LIN {X 0,Y 531.006,Z 455.967,A -85,B 0,C 180,E1 -4200.872,E2 -4200.872} C_VEL
LIN {X 0,Y 531.011,Z 455.964,A -85,B 0,C 180,E1 -4203.258,E2 -4203.258} C_VEL
LIN {X 0,Y 530.999,Z 456.014,A -85,B 0,C 180,E1 -4205.596,E2 -4205.596} C_VEL
LIN {X 0,Y 532.647,Z 464.711,A -85,B 0,C 180,E1 -4207.095,E2 -4207.095} C_VEL
LIN {X 0,Y 532.18,Z 482.462,A -85,B 0,C 180,E1 -4209.92,E2 -4209.92} C_VEL
LIN {X 0,Y 531.695,Z 501.444,A -85,B 0,C 180,E1 -4212.897,E2 -4212.897} C_VEL
LIN {X 0,Y 531.421,Z 515.316,A -85,B 0,C 180,E1 -4215.054,E2 -4215.054} C_VEL
LIN {X 0,Y 532.885,Z 524.969,A -85,B 0,C 180,E1 -4215.236,E2 -4215.236} C_VEL
LIN {X 0,Y 532.487,Z 624.081,A -85,B 0,C 180,E1 -4216.598,E2 -4216.598} C_VEL
LIN {X 0,Y 532.307,Z 637.145,A -85,B 0,C 180,E1 -4216.934,E2 -4216.934} C_VEL
LIN {X 0,Y 532.081,Z 649.714,A -85,B 0,C 180,E1 -4217.413,E2 -4217.413} C_VEL
LIN {X 0,Y 531.842,Z 661.515,A -85,B 0,C 180,E1 -4218.027,E2 -4218.027} C_VEL
LIN {X 0,Y 531.577,Z 672.421,A -85,B 0,C 180,E1 -4218.756,E2 -4218.756} C_VEL
LIN {X 0,Y 531.264,Z 682.786,A -85,B 0,C 180,E1 -4219.617,E2 -4219.617} C_VEL
LIN {X 0,Y 531.07,Z 691.257,A -85,B 0,C 180,E1 -4220.479,E2 -4220.479} C_VEL
LIN {X 0,Y 530.852,Z 700.523,A -85,B 0,C 180,E1 -4221.627,E2 -4221.627} C_VEL
LIN {X 0,Y 530.672,Z 707.981,A -85,B 0,C 180,E1 -4222.773,E2 -4222.773} C_VEL
LIN {X 0,Y 530.606,Z 713.97,A -85,B 0,C 180,E1 -4223.918,E2 -4223.918} C_VEL
LIN {X 0,Y 530.459,Z 718.708,A -85,B 0,C 180,E1 -4225.061,E2 -4225.061} C_VEL
LIN {X 0,Y 530.516,Z 722.337,A -85,B 0,C 180,E1 -4226.203,E2 -4226.203} C_VEL
LIN {X 0,Y 530.457,Z 724.213,A -85,B 0,C 180,E1 -4226.963,E2 -4226.963} C_VEL
LIN {X 0,Y 530.411,Z 725.631,A -85,B 0,C 180,E1 -4227.723,E2 -4227.723} C_VEL
LIN {X 0,Y 530.344,Z 727.258,A -85,B 0,C 180,E1 -4229.242,E2 -4229.242} C_VEL
LIN {X 0,Y 530.343,Z 727.497,A -85,B 0,C 180,E1 -4230.001,E2 -4230.001} C_VEL
LIN {X 0,Y 530.344,Z 727.313,A -85,B 0,C 180,E1 -4230.76,E2 -4230.76} C_VEL
LIN {X 0,Y 530.411,Z 725.758,A -85,B 0,C 180,E1 -4232.279,E2 -4232.279} C_VEL
LIN {X 0,Y 530.458,Z 724.396,A -85,B 0,C 180,E1 -4233.039,E2 -4233.039} C_VEL
LIN {X 0,Y 530.523,Z 721.517,A -85,B 0,C 180,E1 -4234.179,E2 -4234.179} C_VEL
LIN {X 0,Y 530.524,Z 717.614,A -85,B 0,C 180,E1 -4235.322,E2 -4235.322} C_VEL
LIN {X 0,Y 530.594,Z 712.029,A -85,B 0,C 180,E1 -4236.577,E2 -4236.577} C_VEL
LIN {X 0,Y 530.759,Z 705.018,A -85,B 0,C 180,E1 -4237.801,E2 -4237.801} C_VEL
LIN {X 0,Y 530.903,Z 696.833,A -85,B 0,C 180,E1 -4238.949,E2 -4238.949} C_VEL
LIN {X 0,Y 531.112,Z 688.547,A -85,B 0,C 180,E1 -4239.906,E2 -4239.906} C_VEL
LIN {X 0,Y 531.419,Z 678.357,A -85,B 0,C 180,E1 -4240.864,E2 -4240.864} C_VEL
LIN {X 0,Y 531.749,Z 666.673,A -85,B 0,C 180,E1 -4241.739,E2 -4241.739} C_VEL
LIN {X 0,Y 531.952,Z 655.511,A -85,B 0,C 180,E1 -4242.398,E2 -4242.398} C_VEL
LIN {X 0,Y 532.204,Z 642.456,A -85,B 0,C 180,E1 -4242.974,E2 -4242.974} C_VEL
LIN {X 0,Y 532.414,Z 629.216,A -85,B 0,C 180,E1 -4243.381,E2 -4243.381} C_VEL
LIN {X 0,Y 532.569,Z 616.016,A -85,B 0,C 180,E1 -4243.62,E2 -4243.62} C_VEL
LIN {X 0,Y 532.812,Z 523.746,A -85,B 0,C 180,E1 -4244.872,E2 -4244.872} C_VEL
LIN {X 0,Y 531.432,Z 515.327,A -85,B 0,C 180,E1 -4245.033,E2 -4245.033} C_VEL
LIN {X 0,Y 531.931,Z 493.174,A -85,B 0,C 180,E1 -4248.488,E2 -4248.488} C_VEL
LIN {X 0,Y 532.405,Z 474.148,A -85,B 0,C 180,E1 -4251.489,E2 -4251.489} C_VEL
LIN {X 0,Y 532.598,Z 463.987,A -85,B 0,C 180,E1 -4253.115,E2 -4253.115} C_VEL
LIN {X 0,Y 531.023,Z 455.965,A -85,B 0,C 180,E1 -4254.535,E2 -4254.535} C_VEL
LIN {X 0,Y 531.022,Z 455.969,A -85,B 0,C 180,E1 -4257.596,E2 -4257.596} C_VEL
LIN {X 0,Y 530.981,Z 455.968,A -85,B 0,C 180,E1 -4260.646,E2 -4260.646} C_VEL
LIN {X 0,Y 530.993,Z 455.97,A -85,B 0,C 180,E1 -4263.773,E2 -4263.773} C_VEL
LIN {X 0,Y 530.961,Z 455.967,A -85,B 0,C 180,E1 -4266.559,E2 -4266.559} C_VEL
LIN {X 0,Y 530.996,Z 455.967,A -85,B 0,C 180,E1 -4269.443,E2 -4269.443} C_VEL
LIN {X 0,Y 530.99,Z 455.964,A -85,B 0,C 180,E1 -4272.456,E2 -4272.456} C_VEL
LIN {X 0,Y 530.99,Z 455.97,A -85,B 0,C 180,E1 -4275.621,E2 -4275.621} C_VEL
LIN {X 0,Y 530.999,Z 455.961,A -85,B 0,C 180,E1 -4278.565,E2 -4278.565} C_VEL
LIN {X 0,Y 530.963,Z 455.972,A -85,B 0,C 180,E1 -4281.53,E2 -4281.53} C_VEL
LIN {X 0,Y 530.988,Z 455.964,A -85,B 0,C 180,E1 -4284.382,E2 -4284.382} C_VEL
LIN {X 0,Y 530.976,Z 455.966,A -85,B 0,C 180,E1 -4287.134,E2 -4287.134} C_VEL
LIN {X 0,Y 530.976,Z 455.973,A -85,B 0,C 180,E1 -4289.803,E2 -4289.803} C_VEL
LIN {X 0,Y 531.018,Z 455.961,A -85,B 0,C 180,E1 -4292.468,E2 -4292.468} C_VEL
LIN {X 0,Y 531.061,Z 456.072,A -85,B 0,C 180,E1 -4294.997,E2 -4294.997} C_VEL
LIN {X 0,Y 532.61,Z 464.294,A -85,B 0,C 180,E1 -4296.268,E2 -4296.268} C_VEL
LIN {X 0,Y 532.339,Z 481.085,A -85,B 0,C 180,E1 -4298.712,E2 -4298.712} C_VEL
LIN {X 0,Y 531.898,Z 502.756,A -85,B 0,C 180,E1 -4301.861,E2 -4301.861} C_VEL
LIN {X 0,Y 531.491,Z 524.306,A -85,B 0,C 180,E1 -4305.003,E2 -4305.003} C_VEL
LIN {X 0,Y 531.503,Z 525.159,A -85,B 0,C 180,E1 -4305.103,E2 -4305.103} C_VEL
LIN {X 0,Y 532.808,Z 533.582,A -85,B 0,C 180,E1 -4305.258,E2 -4305.258} C_VEL
LIN {X 0,Y 532.385,Z 632.475,A -85,B 0,C 180,E1 -4306.619,E2 -4306.619} C_VEL
LIN {X 0,Y 532.252,Z 643.791,A -85,B 0,C 180,E1 -4306.882,E2 -4306.882} C_VEL
LIN {X 0,Y 532.047,Z 656.313,A -85,B 0,C 180,E1 -4307.314,E2 -4307.314} C_VEL
LIN {X 0,Y 531.83,Z 669.019,A -85,B 0,C 180,E1 -4307.932,E2 -4307.932} C_VEL
LIN {X 0,Y 531.631,Z 679.052,A -85,B 0,C 180,E1 -4308.563,E2 -4308.563} C_VEL
LIN {X 0,Y 531.377,Z 687.856,A -85,B 0,C 180,E1 -4309.233,E2 -4309.233} C_VEL
LIN {X 0,Y 531.202,Z 695.315,A -85,B 0,C 180,E1 -4309.904,E2 -4309.904} C_VEL
LIN {X 0,Y 531.026,Z 702.592,A -85,B 0,C 180,E1 -4310.67,E2 -4310.67} C_VEL
LIN {X 0,Y 530.847,Z 710.181,A -85,B 0,C 180,E1 -4311.626,E2 -4311.626} C_VEL
LIN {X 0,Y 530.687,Z 716.517,A -85,B 0,C 180,E1 -4312.581,E2 -4312.581} C_VEL
LIN {X 0,Y 530.551,Z 722.563,A -85,B 0,C 180,E1 -4313.695,E2 -4313.695} C_VEL
LIN {X 0,Y 530.524,Z 726.919,A -85,B 0,C 180,E1 -4314.679,E2 -4314.679} C_VEL
LIN {X 0,Y 530.523,Z 730.899,A -85,B 0,C 180,E1 -4315.822,E2 -4315.822} C_VEL
LIN {X 0,Y 530.458,Z 733.85,A -85,B 0,C 180,E1 -4316.962,E2 -4316.962} C_VEL
LIN {X 0,Y 530.411,Z 735.354,A -85,B 0,C 180,E1 -4317.722,E2 -4317.722} C_VEL
LIN {X 0,Y 530.344,Z 736.92,A -85,B 0,C 180,E1 -4319.241,E2 -4319.241} C_VEL
LIN {X 0,Y 530.343,Z 737.208,A -85,B 0,C 180,E1 -4320,E2 -4320} C_VEL
LIN {X 0,Y 530.361,Z 736.404,A -85,B 0,C 180,E1 -4321.519,E2 -4321.519} C_VEL
LIN {X 0,Y 530.41,Z 735.49,A -85,B 0,C 180,E1 -4322.278,E2 -4322.278} C_VEL
LIN {X 0,Y 530.516,Z 732.244,A -85,B 0,C 180,E1 -4323.798,E2 -4323.798} C_VEL
LIN {X 0,Y 530.459,Z 728.685,A -85,B 0,C 180,E1 -4324.94,E2 -4324.94} C_VEL
LIN {X 0,Y 530.606,Z 725.794,A -85,B 0,C 180,E1 -4325.701,E2 -4325.701} C_VEL
LIN {X 0,Y 530.644,Z 720.318,A -85,B 0,C 180,E1 -4326.846,E2 -4326.846} C_VEL
LIN {X 0,Y 530.779,Z 713.434,A -85,B 0,C 180,E1 -4327.992,E2 -4327.992} C_VEL
LIN {X 0,Y 530.905,Z 706.468,A -85,B 0,C 180,E1 -4328.948,E2 -4328.948} C_VEL
LIN {X 0,Y 531.091,Z 699.912,A -85,B 0,C 180,E1 -4329.713,E2 -4329.713} C_VEL
LIN {X 0,Y 531.276,Z 691.104,A -85,B 0,C 180,E1 -4330.576,E2 -4330.576} C_VEL
LIN {X 0,Y 531.491,Z 682.944,A -85,B 0,C 180,E1 -4331.247,E2 -4331.247} C_VEL
LIN {X 0,Y 531.712,Z 673.503,A -85,B 0,C 180,E1 -4331.891,E2 -4331.891} C_VEL
LIN {X 0,Y 531.892,Z 664.443,A -85,B 0,C 180,E1 -4332.399,E2 -4332.399} C_VEL
LIN {X 0,Y 532.109,Z 653.571,A -85,B 0,C 180,E1 -4332.878,E2 -4332.878} C_VEL
LIN {X 0,Y 532.259,Z 642.616,A -85,B 0,C 180,E1 -4333.239,E2 -4333.239} C_VEL
LIN {X 0,Y 532.403,Z 631.966,A -85,B 0,C 180,E1 -4333.478,E2 -4333.478} C_VEL
LIN {X 0,Y 532.71,Z 532.707,A -85,B 0,C 180,E1 -4334.847,E2 -4334.847} C_VEL
LIN {X 0,Y 531.443,Z 524.939,A -85,B 0,C 180,E1 -4334.999,E2 -4334.999} C_VEL
LIN {X 0,Y 531.875,Z 505.036,A -85,B 0,C 180,E1 -4337.938,E2 -4337.938} C_VEL
LIN {X 0,Y 532.203,Z 485.232,A -85,B 0,C 180,E1 -4340.717,E2 -4340.717} C_VEL
LIN {X 0,Y 532.417,Z 472.579,A -85,B 0,C 180,E1 -4342.508,E2 -4342.508} C_VEL
LIN {X 0,Y 532.451,Z 463.714,A -85,B 0,C 180,E1 -4343.739,E2 -4343.739} C_VEL
LIN {X 0,Y 531.068,Z 455.96,A -85,B 0,C 180,E1 -4344.871,E2 -4344.871} C_VEL
LIN {X 0,Y 531.02,Z 455.963,A -85,B 0,C 180,E1 -4347.595,E2 -4347.595} C_VEL
LIN {X 0,Y 530.979,Z 455.97,A -85,B 0,C 180,E1 -4350.645,E2 -4350.645} C_VEL
LIN {X 0,Y 530.996,Z 455.968,A -85,B 0,C 180,E1 -4353.772,E2 -4353.772} C_VEL
LIN {X 0,Y 530.974,Z 455.968,A -85,B 0,C 180,E1 -4356.557,E2 -4356.557} C_VEL
LIN {X 0,Y 530.983,Z 455.972,A -85,B 0,C 180,E1 -4359.853,E2 -4359.853} C_VEL
LIN {X 0,Y 530.982,Z 455.967,A -85,B 0,C 180,E1 -4362.456,E2 -4362.456} C_VEL
LIN {X 0,Y 530.987,Z 455.97,A -85,B 0,C 180,E1 -4365.621,E2 -4365.621} C_VEL
LIN {X 0,Y 531.001,Z 455.962,A -85,B 0,C 180,E1 -4368.564,E2 -4368.564} C_VEL
LIN {X 0,Y 530.962,Z 455.973,A -85,B 0,C 180,E1 -4371.529,E2 -4371.529} C_VEL
LIN {X 0,Y 530.959,Z 455.968,A -85,B 0,C 180,E1 -4374.379,E2 -4374.379} C_VEL
LIN {X 0,Y 530.972,Z 455.971,A -85,B 0,C 180,E1 -4377.133,E2 -4377.133} C_VEL
LIN {X 0,Y 530.974,Z 455.971,A -85,B 0,C 180,E1 -4379.803,E2 -4379.803} C_VEL
LIN {X 0,Y 531.02,Z 455.963,A -85,B 0,C 180,E1 -4382.466,E2 -4382.466} C_VEL
LIN {X 0,Y 531.013,Z 456.03,A -85,B 0,C 180,E1 -4383.767,E2 -4383.767} C_VEL
LIN {X 0,Y 533.679,Z 467.602,A -85,B 0,C 180,E1 -4385.321,E2 -4385.321} C_VEL
LIN {X 0,Y 533.111,Z 489.338,A -85,B 0,C 180,E1 -4387.931,E2 -4387.931} C_VEL
LIN {X 0,Y 532.417,Z 514.942,A -85,B 0,C 180,E1 -4390.93,E2 -4390.93} C_VEL
LIN {X 0,Y 532.244,Z 523.261,A -85,B 0,C 180,E1 -4391.895,E2 -4391.895} C_VEL
LIN {X 0,Y 533.886,Z 534.58,A -85,B 0,C 180,E1 -4392.117,E2 -4392.117} C_VEL
LIN {X 0,Y 533.234,Z 661.903,A -85,B 0,C 180,E1 -4393.857,E2 -4393.857} C_VEL
LIN {X 0,Y 532.984,Z 676.417,A -85,B 0,C 180,E1 -4394.205,E2 -4394.205} C_VEL
LIN {X 0,Y 532.791,Z 690.417,A -85,B 0,C 180,E1 -4394.702,E2 -4394.702} C_VEL
LIN {X 0,Y 532.51,Z 702.779,A -85,B 0,C 180,E1 -4395.281,E2 -4395.281} C_VEL
LIN {X 0,Y 532.115,Z 715.658,A -85,B 0,C 180,E1 -4396.051,E2 -4396.051} C_VEL
LIN {X 0,Y 531.815,Z 727.295,A -85,B 0,C 180,E1 -4396.919,E2 -4396.919} C_VEL
LIN {X 0,Y 531.465,Z 738.305,A -85,B 0,C 180,E1 -4397.916,E2 -4397.916} C_VEL
LIN {X 0,Y 531.236,Z 747.698,A -85,B 0,C 180,E1 -4398.94,E2 -4398.94} C_VEL
LIN {X 0,Y 530.936,Z 756.55,A -85,B 0,C 180,E1 -4400.09,E2 -4400.09} C_VEL
LIN {X 0,Y 530.776,Z 765.028,A -85,B 0,C 180,E1 -4401.432,E2 -4401.432} C_VEL
LIN {X 0,Y 530.587,Z 771.859,A -85,B 0,C 180,E1 -4402.77,E2 -4402.77} C_VEL
LIN {X 0,Y 530.585,Z 777.957,A -85,B 0,C 180,E1 -4404.298,E2 -4404.298} C_VEL
LIN {X 0,Y 530.449,Z 781.441,A -85,B 0,C 180,E1 -4405.44,E2 -4405.44} C_VEL
LIN {X 0,Y 530.452,Z 784.831,A -85,B 0,C 180,E1 -4406.961,E2 -4406.961} C_VEL
LIN {X 0,Y 530.356,Z 786.834,A -85,B 0,C 180,E1 -4408.48,E2 -4408.48} C_VEL
LIN {X 0,Y 530.341,Z 787.5,A -85,B 0,C 180,E1 -4409.999,E2 -4409.999} C_VEL
LIN {X 0,Y 530.356,Z 786.837,A -85,B 0,C 180,E1 -4411.518,E2 -4411.518} C_VEL
LIN {X 0,Y 530.452,Z 784.838,A -85,B 0,C 180,E1 -4413.037,E2 -4413.037} C_VEL
LIN {X 0,Y 530.449,Z 781.45,A -85,B 0,C 180,E1 -4414.559,E2 -4414.559} C_VEL
LIN {X 0,Y 530.545,Z 776.571,A -85,B 0,C 180,E1 -4416.082,E2 -4416.082} C_VEL
LIN {X 0,Y 530.639,Z 770.059,A -85,B 0,C 180,E1 -4417.61,E2 -4417.61} C_VEL
LIN {X 0,Y 530.809,Z 762.81,A -85,B 0,C 180,E1 -4418.949,E2 -4418.949} C_VEL
LIN {X 0,Y 531.023,Z 753.83,A -85,B 0,C 180,E1 -4420.291,E2 -4420.291} C_VEL
LIN {X 0,Y 531.336,Z 744.403,A -85,B 0,C 180,E1 -4421.443,E2 -4421.443} C_VEL
LIN {X 0,Y 531.595,Z 733.963,A -85,B 0,C 180,E1 -4422.502,E2 -4422.502} C_VEL
LIN {X 0,Y 531.955,Z 722.441,A -85,B 0,C 180,E1 -4423.464,E2 -4423.464} C_VEL
LIN {X 0,Y 532.338,Z 709.642,A -85,B 0,C 180,E1 -4424.331,E2 -4424.331} C_VEL
LIN {X 0,Y 532.616,Z 697,A -85,B 0,C 180,E1 -4425.007,E2 -4425.007} C_VEL
LIN {X 0,Y 532.889,Z 683.114,A -85,B 0,C 180,E1 -4425.578,E2 -4425.578} C_VEL
LIN {X 0,Y 533.163,Z 668.658,A -85,B 0,C 180,E1 -4426.001,E2 -4426.001} C_VEL
LIN {X 0,Y 533.291,Z 654.28,A -85,B 0,C 180,E1 -4426.262,E2 -4426.262} C_VEL
LIN {X 0,Y 533.824,Z 533.283,A -85,B 0,C 180,E1 -4427.902,E2 -4427.902} C_VEL
LIN {X 0,Y 532.256,Z 523.34,A -85,B 0,C 180,E1 -4428.095,E2 -4428.095} C_VEL
LIN {X 0,Y 532.905,Z 496.157,A -85,B 0,C 180,E1 -4431.263,E2 -4431.263} C_VEL
LIN {X 0,Y 533.655,Z 471.16,A -85,B 0,C 180,E1 -4434.239,E2 -4434.239} C_VEL
LIN {X 0,Y 533.728,Z 467.421,A -85,B 0,C 180,E1 -4434.691,E2 -4434.691} C_VEL
LIN {X 0,Y 531.003,Z 455.969,A -85,B 0,C 180,E1 -4436.26,E2 -4436.26} C_VEL
LIN {X 0,Y 530.997,Z 455.964,A -85,B 0,C 180,E1 -4439.32,E2 -4439.32} C_VEL
LIN {X 0,Y 530.977,Z 455.967,A -85,B 0,C 180,E1 -4442.102,E2 -4442.102} C_VEL
LIN {X 0,Y 530.986,Z 455.963,A -85,B 0,C 180,E1 -4444.853,E2 -4444.853} C_VEL
LIN {X 0,Y 530.962,Z 455.967,A -85,B 0,C 180,E1 -4447.506,E2 -4447.506} C_VEL
LIN {X 0,Y 531.022,Z 455.965,A -85,B 0,C 180,E1 -4450.427,E2 -4450.427} C_VEL
LIN {X 0,Y 530.962,Z 455.966,A -85,B 0,C 180,E1 -4453.493,E2 -4453.493} C_VEL
LIN {X 0,Y 530.959,Z 455.972,A -85,B 0,C 180,E1 -4456.505,E2 -4456.505} C_VEL
LIN {X 0,Y 531.001,Z 455.96,A -85,B 0,C 180,E1 -4459.569,E2 -4459.569} C_VEL
LIN {X 0,Y 530.96,Z 455.972,A -85,B 0,C 180,E1 -4462.576,E2 -4462.576} C_VEL
LIN {X 0,Y 530.996,Z 455.96,A -85,B 0,C 180,E1 -4465.311,E2 -4465.311} C_VEL
LIN {X 0,Y 530.973,Z 455.965,A -85,B 0,C 180,E1 -4468.032,E2 -4468.032} C_VEL
LIN {X 0,Y 530.997,Z 455.967,A -85,B 0,C 180,E1 -4470.87,E2 -4470.87} C_VEL
LIN {X 0,Y 531.003,Z 455.962,A -85,B 0,C 180,E1 -4473.256,E2 -4473.256} C_VEL
LIN {X 0,Y 530.986,Z 455.962,A -85,B 0,C 180,E1 -4475.957,E2 -4475.957} C_VEL
LIN {X 0,Y 530.992,Z 455.962,A -85,B 0,C 180,E1 -4479.062,E2 -4479.062} C_VEL
LIN {X 0,Y 531.005,Z 455.965,A -85,B 0,C 180,E1 -4482.277,E2 -4482.277} C_VEL
LIN {X 0,Y 531.008,Z 455.96,A -85,B 0,C 180,E1 -4485.436,E2 -4485.436} C_VEL
LIN {X 0,Y 531.036,Z 455.963,A -85,B 0,C 180,E1 -4488.55,E2 -4488.55} C_VEL
LIN {X 0,Y 531.051,Z 455.955,A -85,B 0,C 180,E1 -4491.629,E2 -4491.629} C_VEL
LIN {X 0,Y 531.132,Z 455.953,A -85,B 0,C 180,E1 -4494.685,E2 -4494.685} C_VEL
LIN {X 0,Y 531.13,Z 455.944,A -85,B 0,C 180,E1 -4497.725,E2 -4497.725} C_VEL
LIN {X 0,Y 531.146,Z 455.95,A -85,B 0,C 180,E1 -4500.758,E2 -4500.758} C_VEL
LIN {X 0,Y 531.101,Z 455.948,A -85,B 0,C 180,E1 -4503.034,E2 -4503.034} C_VEL
LIN {X 0,Y 531.074,Z 455.955,A -85,B 0,C 180,E1 -4506.077,E2 -4506.077} C_VEL
LIN {X 0,Y 531.026,Z 455.959,A -85,B 0,C 180,E1 -4509.138,E2 -4509.138} C_VEL
LIN {X 0,Y 531.03,Z 455.962,A -85,B 0,C 180,E1 -4512.225,E2 -4512.225} C_VEL
LIN {X 0,Y 530.986,Z 455.963,A -85,B 0,C 180,E1 -4515.35,E2 -4515.35} C_VEL
LIN {X 0,Y 531.006,Z 455.959,A -85,B 0,C 180,E1 -4517.723,E2 -4517.723} C_VEL
LIN {X 0,Y 530.992,Z 455.965,A -85,B 0,C 180,E1 -4520.938,E2 -4520.938} C_VEL
LIN {X 0,Y 530.97,Z 455.97,A -85,B 0,C 180,E1 -4524.225,E2 -4524.225} C_VEL
LIN {X 0,Y 531.003,Z 455.966,A -85,B 0,C 180,E1 -4526.744,E2 -4526.744} C_VEL
LIN {X 0,Y 530.991,Z 455.962,A -85,B 0,C 180,E1 -4529.322,E2 -4529.322} C_VEL
LIN {X 0,Y 530.972,Z 455.968,A -85,B 0,C 180,E1 -4532.104,E2 -4532.104} C_VEL
LIN {X 0,Y 530.984,Z 455.968,A -85,B 0,C 180,E1 -4534.856,E2 -4534.856} C_VEL
LIN {X 0,Y 530.96,Z 455.965,A -85,B 0,C 180,E1 -4537.508,E2 -4537.508} C_VEL
LIN {X 0,Y 531.02,Z 455.967,A -85,B 0,C 180,E1 -4540.43,E2 -4540.43} C_VEL
LIN {X 0,Y 530.955,Z 455.967,A -85,B 0,C 180,E1 -4543.578,E2 -4543.578} C_VEL
LIN {X 0,Y 530.284,Z 456.057,A -85,B 0,C 180,E1 -4544.212,E2 -4544.212} C_VEL
LIN {X 0,Y 527.438,Z 456.413,A -85,B 0,C 180,E1 -4545.241,E2 -4545.241} C_VEL
LIN {X 0,Y 525.035,Z 456.713,A -85,B 0,C 180,E1 -4546.069,E2 -4546.069} C_VEL
LIN {X 0,Y 524.002,Z 456.84,A -85,B 0,C 180,E1 -4546.709,E2 -4546.709} C_VEL
LIN {X 0,Y 523.917,Z 456.847,A -85,B 0,C 180,E1 -4546.925,E2 -4546.925} C_VEL
LIN {X 0,Y 523.974,Z 456.839,A -85,B 0,C 180,E1 -4549.925,E2 -4549.925} C_VEL
LIN {X 0,Y 523.908,Z 456.847,A -85,B 0,C 180,E1 -4552.87,E2 -4552.87} C_VEL
LIN {X 0,Y 523.943,Z 456.842,A -85,B 0,C 180,E1 -4555.712,E2 -4555.712} C_VEL
LIN {X 0,Y 523.931,Z 456.848,A -85,B 0,C 180,E1 -4558.458,E2 -4558.458} C_VEL
LIN {X 0,Y 523.95,Z 456.844,A -85,B 0,C 180,E1 -4561.127,E2 -4561.127} C_VEL
LIN {X 0,Y 523.985,Z 456.842,A -85,B 0,C 180,E1 -4563.981,E2 -4563.981} C_VEL
LIN {X 0,Y 523.985,Z 456.933,A -85,B 0,C 180,E1 -4565.379,E2 -4565.379} C_VEL
LIN {X 0,Y 525.753,Z 466.105,A -85,B 0,C 180,E1 -4566.985,E2 -4566.985} C_VEL
LIN {X 0,Y 525.292,Z 482.605,A -85,B 0,C 180,E1 -4569.645,E2 -4569.645} C_VEL
LIN {X 0,Y 524.777,Z 501.605,A -85,B 0,C 180,E1 -4572.665,E2 -4572.665} C_VEL
LIN {X 0,Y 524.451,Z 515.395,A -85,B 0,C 180,E1 -4574.829,E2 -4574.829} C_VEL
LIN {X 0,Y 526.097,Z 525.449,A -85,B 0,C 180,E1 -4575.02,E2 -4575.02} C_VEL
LIN {X 0,Y 525.687,Z 623.589,A -85,B 0,C 180,E1 -4576.372,E2 -4576.372} C_VEL
LIN {X 0,Y 525.489,Z 636.208,A -85,B 0,C 180,E1 -4576.687,E2 -4576.687} C_VEL
LIN {X 0,Y 525.241,Z 649.671,A -85,B 0,C 180,E1 -4577.197,E2 -4577.197} C_VEL
LIN {X 0,Y 524.976,Z 660.656,A -85,B 0,C 180,E1 -4577.762,E2 -4577.762} C_VEL
LIN {X 0,Y 524.713,Z 671.91,A -85,B 0,C 180,E1 -4578.509,E2 -4578.509} C_VEL
LIN {X 0,Y 524.344,Z 682.423,A -85,B 0,C 180,E1 -4579.381,E2 -4579.381} C_VEL
LIN {X 0,Y 524.111,Z 691.886,A -85,B 0,C 180,E1 -4580.352,E2 -4580.352} C_VEL
LIN {X 0,Y 523.893,Z 699.65,A -85,B 0,C 180,E1 -4581.321,E2 -4581.321} C_VEL
LIN {X 0,Y 523.66,Z 707.249,A -85,B 0,C 180,E1 -4582.482,E2 -4582.482} C_VEL
LIN {X 0,Y 523.542,Z 714.234,A -85,B 0,C 180,E1 -4583.836,E2 -4583.836} C_VEL
LIN {X 0,Y 523.383,Z 718.899,A -85,B 0,C 180,E1 -4584.994,E2 -4584.994} C_VEL
LIN {X 0,Y 523.443,Z 722.463,A -85,B 0,C 180,E1 -4586.152,E2 -4586.152} C_VEL
LIN {X 0,Y 523.367,Z 724.313,A -85,B 0,C 180,E1 -4586.922,E2 -4586.922} C_VEL
LIN {X 0,Y 523.335,Z 725.709,A -85,B 0,C 180,E1 -4587.692,E2 -4587.692} C_VEL
LIN {X 0,Y 523.25,Z 727.316,A -85,B 0,C 180,E1 -4589.231,E2 -4589.231} C_VEL
LIN {X 0,Y 523.247,Z 727.551,A -85,B 0,C 180,E1 -4590.001,E2 -4590.001} C_VEL
LIN {X 0,Y 523.25,Z 727.369,A -85,B 0,C 180,E1 -4590.771,E2 -4590.771} C_VEL
LIN {X 0,Y 523.335,Z 725.831,A -85,B 0,C 180,E1 -4592.31,E2 -4592.31} C_VEL
LIN {X 0,Y 523.368,Z 724.489,A -85,B 0,C 180,E1 -4593.08,E2 -4593.08} C_VEL
LIN {X 0,Y 523.442,Z 721.651,A -85,B 0,C 180,E1 -4594.236,E2 -4594.236} C_VEL
LIN {X 0,Y 523.463,Z 717.811,A -85,B 0,C 180,E1 -4595.394,E2 -4595.394} C_VEL
LIN {X 0,Y 523.518,Z 712.761,A -85,B 0,C 180,E1 -4596.575,E2 -4596.575} C_VEL
LIN {X 0,Y 523.682,Z 706.637,A -85,B 0,C 180,E1 -4597.713,E2 -4597.713} C_VEL
LIN {X 0,Y 523.895,Z 698.849,A -85,B 0,C 180,E1 -4598.875,E2 -4598.875} C_VEL
LIN {X 0,Y 524.152,Z 689.17,A -85,B 0,C 180,E1 -4600.039,E2 -4600.039} C_VEL
LIN {X 0,Y 524.486,Z 679.066,A -85,B 0,C 180,E1 -4601.009,E2 -4601.009} C_VEL
LIN {X 0,Y 524.86,Z 667.864,A -85,B 0,C 180,E1 -4601.867,E2 -4601.867} C_VEL
LIN {X 0,Y 525.079,Z 656.426,A -85,B 0,C 180,E1 -4602.563,E2 -4602.563} C_VEL
LIN {X 0,Y 525.355,Z 644.892,A -85,B 0,C 180,E1 -4603.097,E2 -4603.097} C_VEL
LIN {X 0,Y 525.559,Z 632.511,A -85,B 0,C 180,E1 -4603.51,E2 -4603.51} C_VEL
LIN {X 0,Y 525.728,Z 619.999,A -85,B 0,C 180,E1 -4603.776,E2 -4603.776} C_VEL
LIN {X 0,Y 525.992,Z 524.359,A -85,B 0,C 180,E1 -4605.084,E2 -4605.084} C_VEL
LIN {X 0,Y 524.449,Z 515.252,A -85,B 0,C 180,E1 -4605.283,E2 -4605.283} C_VEL
LIN {X 0,Y 524.979,Z 494.705,A -85,B 0,C 180,E1 -4608.519,E2 -4608.519} C_VEL
LIN {X 0,Y 525.362,Z 478.073,A -85,B 0,C 180,E1 -4611.174,E2 -4611.174} C_VEL
LIN {X 0,Y 525.773,Z 466.631,A -85,B 0,C 180,E1 -4613.017,E2 -4613.017} C_VEL
LIN {X 0,Y 523.981,Z 456.843,A -85,B 0,C 180,E1 -4614.729,E2 -4614.729} C_VEL
LIN {X 0,Y 523.985,Z 456.847,A -85,B 0,C 180,E1 -4617.719,E2 -4617.719} C_VEL
LIN {X 0,Y 523.951,Z 456.844,A -85,B 0,C 180,E1 -4620.855,E2 -4620.855} C_VEL
LIN {X 0,Y 523.965,Z 456.846,A -85,B 0,C 180,E1 -4623.735,E2 -4623.735} C_VEL
LIN {X 0,Y 523.909,Z 456.846,A -85,B 0,C 180,E1 -4626.402,E2 -4626.402} C_VEL
LIN {X 0,Y 523.929,Z 456.843,A -85,B 0,C 180,E1 -4629.085,E2 -4629.085} C_VEL
LIN {X 0,Y 523.964,Z 456.842,A -85,B 0,C 180,E1 -4632.119,E2 -4632.119} C_VEL
LIN {X 0,Y 523.961,Z 456.841,A -85,B 0,C 180,E1 -4635.309,E2 -4635.309} C_VEL
LIN {X 0,Y 523.961,Z 456.837,A -85,B 0,C 180,E1 -4638.69,E2 -4638.69} C_VEL
LIN {X 0,Y 523.923,Z 456.844,A -85,B 0,C 180,E1 -4641.081,E2 -4641.081} C_VEL
LIN {X 0,Y 523.935,Z 456.849,A -85,B 0,C 180,E1 -4643.828,E2 -4643.828} C_VEL
LIN {X 0,Y 523.949,Z 456.84,A -85,B 0,C 180,E1 -4646.636,E2 -4646.636} C_VEL
LIN {X 0,Y 523.961,Z 456.843,A -85,B 0,C 180,E1 -4649.356,E2 -4649.356} C_VEL
LIN {X 0,Y 523.983,Z 456.839,A -85,B 0,C 180,E1 -4652.282,E2 -4652.282} C_VEL
LIN {X 0,Y 524.034,Z 456.99,A -85,B 0,C 180,E1 -4654.824,E2 -4654.824} C_VEL
LIN {X 0,Y 525.683,Z 465.511,A -85,B 0,C 180,E1 -4656.151,E2 -4656.151} C_VEL
LIN {X 0,Y 525.437,Z 479.564,A -85,B 0,C 180,E1 -4658.212,E2 -4658.212} C_VEL
LIN {X 0,Y 525.055,Z 497.625,A -85,B 0,C 180,E1 -4660.856,E2 -4660.856} C_VEL
LIN {X 0,Y 524.631,Z 518.142,A -85,B 0,C 180,E1 -4663.861,E2 -4663.861} C_VEL
LIN {X 0,Y 524.523,Z 525.245,A -85,B 0,C 180,E1 -4664.9,E2 -4664.9} C_VEL
LIN {X 0,Y 525.954,Z 534.643,A -85,B 0,C 180,E1 -4665.081,E2 -4665.081} C_VEL
LIN {X 0,Y 525.444,Z 633.269,A -85,B 0,C 180,E1 -4666.463,E2 -4666.463} C_VEL
LIN {X 0,Y 525.332,Z 646.029,A -85,B 0,C 180,E1 -4666.78,E2 -4666.78} C_VEL
LIN {X 0,Y 525.05,Z 659.504,A -85,B 0,C 180,E1 -4667.29,E2 -4667.29} C_VEL
LIN {X 0,Y 524.795,Z 671.704,A -85,B 0,C 180,E1 -4667.929,E2 -4667.929} C_VEL
LIN {X 0,Y 524.571,Z 681.798,A -85,B 0,C 180,E1 -4668.602,E2 -4668.602} C_VEL
LIN {X 0,Y 524.277,Z 692.414,A -85,B 0,C 180,E1 -4669.476,E2 -4669.476} C_VEL
LIN {X 0,Y 524.012,Z 702.751,A -85,B 0,C 180,E1 -4670.544,E2 -4670.544} C_VEL
LIN {X 0,Y 523.825,Z 710.34,A -85,B 0,C 180,E1 -4671.513,E2 -4671.513} C_VEL
LIN {X 0,Y 523.629,Z 717.75,A -85,B 0,C 180,E1 -4672.674,E2 -4672.674} C_VEL
LIN {X 0,Y 523.504,Z 723.712,A -85,B 0,C 180,E1 -4673.834,E2 -4673.834} C_VEL
LIN {X 0,Y 523.463,Z 727.01,A -85,B 0,C 180,E1 -4674.607,E2 -4674.607} C_VEL
LIN {X 0,Y 523.442,Z 730.957,A -85,B 0,C 180,E1 -4675.765,E2 -4675.765} C_VEL
LIN {X 0,Y 523.368,Z 733.882,A -85,B 0,C 180,E1 -4676.921,E2 -4676.921} C_VEL
LIN {X 0,Y 523.335,Z 735.374,A -85,B 0,C 180,E1 -4677.691,E2 -4677.691} C_VEL
LIN {X 0,Y 523.251,Z 736.924,A -85,B 0,C 180,E1 -4679.23,E2 -4679.23} C_VEL
LIN {X 0,Y 523.247,Z 737.213,A -85,B 0,C 180,E1 -4680,E2 -4680} C_VEL
LIN {X 0,Y 523.275,Z 736.413,A -85,B 0,C 180,E1 -4681.539,E2 -4681.539} C_VEL
LIN {X 0,Y 523.334,Z 735.509,A -85,B 0,C 180,E1 -4682.309,E2 -4682.309} C_VEL
LIN {X 0,Y 523.444,Z 732.289,A -85,B 0,C 180,E1 -4683.849,E2 -4683.849} C_VEL
LIN {X 0,Y 523.383,Z 728.768,A -85,B 0,C 180,E1 -4685.007,E2 -4685.007} C_VEL
LIN {X 0,Y 523.537,Z 725.884,A -85,B 0,C 180,E1 -4685.778,E2 -4685.778} C_VEL
LIN {X 0,Y 523.61,Z 719.361,A -85,B 0,C 180,E1 -4687.132,E2 -4687.132} C_VEL
LIN {X 0,Y 523.748,Z 713.594,A -85,B 0,C 180,E1 -4688.1,E2 -4688.1} C_VEL
LIN {X 0,Y 523.869,Z 706.649,A -85,B 0,C 180,E1 -4689.069,E2 -4689.069} C_VEL
LIN {X 0,Y 524.099,Z 698.24,A -85,B 0,C 180,E1 -4690.039,E2 -4690.039} C_VEL
LIN {X 0,Y 524.378,Z 689.049,A -85,B 0,C 180,E1 -4690.912,E2 -4690.912} C_VEL
LIN {X 0,Y 524.699,Z 677.592,A -85,B 0,C 180,E1 -4691.791,E2 -4691.791} C_VEL
LIN {X 0,Y 524.895,Z 666.262,A -85,B 0,C 180,E1 -4692.468,E2 -4692.468} C_VEL
LIN {X 0,Y 525.161,Z 654.625,A -85,B 0,C 180,E1 -4693.002,E2 -4693.002} C_VEL
LIN {X 0,Y 525.363,Z 642.221,A -85,B 0,C 180,E1 -4693.416,E2 -4693.416} C_VEL
LIN {X 0,Y 525.54,Z 629.692,A -85,B 0,C 180,E1 -4693.682,E2 -4693.682} C_VEL
LIN {X 0,Y 525.798,Z 533.176,A -85,B 0,C 180,E1 -4695.039,E2 -4695.039} C_VEL
LIN {X 0,Y 524.507,Z 525.219,A -85,B 0,C 180,E1 -4695.203,E2 -4695.203} C_VEL
LIN {X 0,Y 524.914,Z 505.746,A -85,B 0,C 180,E1 -4698.081,E2 -4698.081} C_VEL
LIN {X 0,Y 525.282,Z 485.236,A -85,B 0,C 180,E1 -4700.971,E2 -4700.971} C_VEL
LIN {X 0,Y 525.522,Z 466.231,A -85,B 0,C 180,E1 -4703.653,E2 -4703.653} C_VEL
LIN {X 0,Y 524.629,Z 460.047,A -85,B 0,C 180,E1 -4704.537,E2 -4704.537} C_VEL
LIN {X 0,Y 524.016,Z 456.838,A -85,B 0,C 180,E1 -4705.017,E2 -4705.017} C_VEL
LIN {X 0,Y 523.975,Z 456.845,A -85,B 0,C 180,E1 -4707.999,E2 -4707.999} C_VEL
LIN {X 0,Y 523.949,Z 456.844,A -85,B 0,C 180,E1 -4710.854,E2 -4710.854} C_VEL
LIN {X 0,Y 523.967,Z 456.844,A -85,B 0,C 180,E1 -4713.735,E2 -4713.735} C_VEL
LIN {X 0,Y 523.928,Z 456.848,A -85,B 0,C 180,E1 -4716.404,E2 -4716.404} C_VEL
LIN {X 0,Y 523.925,Z 456.844,A -85,B 0,C 180,E1 -4719.084,E2 -4719.084} C_VEL
LIN {X 0,Y 523.956,Z 456.846,A -85,B 0,C 180,E1 -4722.119,E2 -4722.119} C_VEL
LIN {X 0,Y 523.95,Z 456.843,A -85,B 0,C 180,E1 -4725.309,E2 -4725.309} C_VEL
LIN {X 0,Y 523.962,Z 456.839,A -85,B 0,C 180,E1 -4728.689,E2 -4728.689} C_VEL
LIN {X 0,Y 523.922,Z 456.845,A -85,B 0,C 180,E1 -4731.08,E2 -4731.08} C_VEL
LIN {X 0,Y 523.905,Z 456.852,A -85,B 0,C 180,E1 -4733.825,E2 -4733.825} C_VEL
LIN {X 0,Y 523.946,Z 456.842,A -85,B 0,C 180,E1 -4736.635,E2 -4736.635} C_VEL
LIN {X 0,Y 523.96,Z 456.847,A -85,B 0,C 180,E1 -4739.355,E2 -4739.355} C_VEL
LIN {X 0,Y 523.983,Z 456.84,A -85,B 0,C 180,E1 -4742.28,E2 -4742.28} C_VEL
LIN {X 0,Y 523.982,Z 456.864,A -85,B 0,C 180,E1 -4743.514,E2 -4743.514} C_VEL
LIN {X 0,Y 526.769,Z 468.646,A -85,B 0,C 180,E1 -4745.126,E2 -4745.126} C_VEL
LIN {X 0,Y 526.517,Z 482.391,A -85,B 0,C 180,E1 -4746.81,E2 -4746.81} C_VEL
LIN {X 0,Y 525.644,Z 509.624,A -85,B 0,C 180,E1 -4750.065,E2 -4750.065} C_VEL
LIN {X 0,Y 525.338,Z 523.258,A -85,B 0,C 180,E1 -4751.675,E2 -4751.675} C_VEL
LIN {X 0,Y 527.039,Z 534.449,A -85,B 0,C 180,E1 -4751.901,E2 -4751.901} C_VEL
LIN {X 0,Y 526.326,Z 662.415,A -85,B 0,C 180,E1 -4753.689,E2 -4753.689} C_VEL
LIN {X 0,Y 526.059,Z 677.127,A -85,B 0,C 180,E1 -4754.058,E2 -4754.058} C_VEL
LIN {X 0,Y 525.802,Z 691.598,A -85,B 0,C 180,E1 -4754.593,E2 -4754.593} C_VEL
LIN {X 0,Y 525.476,Z 705.413,A -85,B 0,C 180,E1 -4755.278,E2 -4755.278} C_VEL
LIN {X 0,Y 525.078,Z 717.817,A -85,B 0,C 180,E1 -4756.058,E2 -4756.058} C_VEL
LIN {X 0,Y 524.725,Z 729.183,A -85,B 0,C 180,E1 -4756.936,E2 -4756.936} C_VEL
LIN {X 0,Y 524.422,Z 740.027,A -85,B 0,C 180,E1 -4757.951,E2 -4757.951} C_VEL
LIN {X 0,Y 524.117,Z 750.782,A -85,B 0,C 180,E1 -4759.179,E2 -4759.179} C_VEL
LIN {X 0,Y 523.864,Z 759.167,A -85,B 0,C 180,E1 -4760.345,E2 -4760.345} C_VEL
LIN {X 0,Y 523.665,Z 767.121,A -85,B 0,C 180,E1 -4761.704,E2 -4761.704} C_VEL
LIN {X 0,Y 523.486,Z 773.524,A -85,B 0,C 180,E1 -4763.059,E2 -4763.059} C_VEL
LIN {X 0,Y 523.452,Z 779.197,A -85,B 0,C 180,E1 -4764.606,E2 -4764.606} C_VEL
LIN {X 0,Y 523.419,Z 783.313,A -85,B 0,C 180,E1 -4766.15,E2 -4766.15} C_VEL
LIN {X 0,Y 523.332,Z 786.001,A -85,B 0,C 180,E1 -4767.69,E2 -4767.69} C_VEL
LIN {X 0,Y 523.247,Z 787.333,A -85,B 0,C 180,E1 -4769.229,E2 -4769.229} C_VEL
LIN {X 0,Y 523.245,Z 787.335,A -85,B 0,C 180,E1 -4770.769,E2 -4770.769} C_VEL
LIN {X 0,Y 523.332,Z 786.007,A -85,B 0,C 180,E1 -4772.308,E2 -4772.308} C_VEL
LIN {X 0,Y 523.418,Z 783.322,A -85,B 0,C 180,E1 -4773.848,E2 -4773.848} C_VEL
LIN {X 0,Y 523.451,Z 779.204,A -85,B 0,C 180,E1 -4775.392,E2 -4775.392} C_VEL
LIN {X 0,Y 523.494,Z 773.53,A -85,B 0,C 180,E1 -4776.939,E2 -4776.939} C_VEL
LIN {X 0,Y 523.663,Z 767.132,A -85,B 0,C 180,E1 -4778.294,E2 -4778.294} C_VEL
LIN {X 0,Y 523.863,Z 759.18,A -85,B 0,C 180,E1 -4779.653,E2 -4779.653} C_VEL
LIN {X 0,Y 524.116,Z 750.798,A -85,B 0,C 180,E1 -4780.819,E2 -4780.819} C_VEL
LIN {X 0,Y 524.426,Z 740.879,A -85,B 0,C 180,E1 -4781.959,E2 -4781.959} C_VEL
LIN {X 0,Y 524.722,Z 729.206,A -85,B 0,C 180,E1 -4783.062,E2 -4783.062} C_VEL
LIN {X 0,Y 525.072,Z 717.85,A -85,B 0,C 180,E1 -4783.94,E2 -4783.94} C_VEL
LIN {X 0,Y 525.47,Z 705.452,A -85,B 0,C 180,E1 -4784.72,E2 -4784.72} C_VEL
LIN {X 0,Y 525.804,Z 691.633,A -85,B 0,C 180,E1 -4785.405,E2 -4785.405} C_VEL
LIN {X 0,Y 526.097,Z 677.442,A -85,B 0,C 180,E1 -4785.93,E2 -4785.93} C_VEL
LIN {X 0,Y 526.284,Z 663.642,A -85,B 0,C 180,E1 -4786.285,E2 -4786.285} C_VEL
LIN {X 0,Y 526.491,Z 637.143,A -85,B 0,C 180,E1 -4786.677,E2 -4786.677} C_VEL
LIN {X 0,Y 527.041,Z 534.663,A -85,B 0,C 180,E1 -4788.096,E2 -4788.096} C_VEL
LIN {X 0,Y 525.343,Z 523.19,A -85,B 0,C 180,E1 -4788.332,E2 -4788.332} C_VEL
LIN {X 0,Y 526.054,Z 495.971,A -85,B 0,C 180,E1 -4791.554,E2 -4791.554} C_VEL
LIN {X 0,Y 526.833,Z 472.178,A -85,B 0,C 180,E1 -4794.426,E2 -4794.426} C_VEL
LIN {X 0,Y 526.777,Z 468.571,A -85,B 0,C 180,E1 -4794.876,E2 -4794.876} C_VEL
LIN {X 0,Y 523.967,Z 456.846,A -85,B 0,C 180,E1 -4796.512,E2 -4796.512} C_VEL
LIN {X 0,Y 523.966,Z 456.84,A -85,B 0,C 180,E1 -4799.326,E2 -4799.326} C_VEL
LIN {X 0,Y 523.936,Z 456.848,A -85,B 0,C 180,E1 -4802.448,E2 -4802.448} C_VEL
LIN {X 0,Y 523.932,Z 456.841,A -85,B 0,C 180,E1 -4805.224,E2 -4805.224} C_VEL
LIN {X 0,Y 523.913,Z 456.847,A -85,B 0,C 180,E1 -4808.1,E2 -4808.1} C_VEL
LIN {X 0,Y 523.963,Z 456.842,A -85,B 0,C 180,E1 -4811.088,E2 -4811.088} C_VEL
LIN {X 0,Y 523.935,Z 456.844,A -85,B 0,C 180,E1 -4814.227,E2 -4814.227} C_VEL
LIN {X 0,Y 523.918,Z 456.85,A -85,B 0,C 180,E1 -4816.833,E2 -4816.833} C_VEL
LIN {X 0,Y 523.97,Z 456.836,A -85,B 0,C 180,E1 -4819.922,E2 -4819.922} C_VEL
LIN {X 0,Y 523.903,Z 456.845,A -85,B 0,C 180,E1 -4822.867,E2 -4822.867} C_VEL
LIN {X 0,Y 523.938,Z 456.838,A -85,B 0,C 180,E1 -4825.71,E2 -4825.71} C_VEL
LIN {X 0,Y 523.923,Z 456.848,A -85,B 0,C 180,E1 -4828.456,E2 -4828.456} C_VEL
LIN {X 0,Y 523.941,Z 456.842,A -85,B 0,C 180,E1 -4831.125,E2 -4831.125} C_VEL
LIN {X 0,Y 523.976,Z 456.837,A -85,B 0,C 180,E1 -4833.979,E2 -4833.979} C_VEL
LIN {X 0,Y 523.926,Z 456.845,A -85,B 0,C 180,E1 -4836.27,E2 -4836.27} C_VEL
LIN {X 0,Y 523.937,Z 456.841,A -85,B 0,C 180,E1 -4838.766,E2 -4838.766} C_VEL
LIN {X 0,Y 523.944,Z 456.842,A -85,B 0,C 180,E1 -4841.221,E2 -4841.221} C_VEL
LIN {X 0,Y 523.931,Z 456.84,A -85,B 0,C 180,E1 -4843.639,E2 -4843.639} C_VEL
LIN {X 0,Y 523.931,Z 456.843,A -85,B 0,C 180,E1 -4846.028,E2 -4846.028} C_VEL
LIN {X 0,Y 524,Z 456.839,A -85,B 0,C 180,E1 -4848.394,E2 -4848.394} C_VEL
LIN {X 0,Y 523.998,Z 456.833,A -85,B 0,C 180,E1 -4851.516,E2 -4851.516} C_VEL
LIN {X 0,Y 524.09,Z 456.829,A -85,B 0,C 180,E1 -4854.614,E2 -4854.614} C_VEL
LIN {X 0,Y 524.102,Z 456.819,A -85,B 0,C 180,E1 -4857.695,E2 -4857.695} C_VEL
LIN {X 0,Y 524.116,Z 456.825,A -85,B 0,C 180,E1 -4860.768,E2 -4860.768} C_VEL
LIN {X 0,Y 524.067,Z 456.824,A -85,B 0,C 180,E1 -4863.075,E2 -4863.075} C_VEL
LIN {X 0,Y 524.036,Z 456.832,A -85,B 0,C 180,E1 -4866.159,E2 -4866.159} C_VEL
LIN {X 0,Y 523.993,Z 456.834,A -85,B 0,C 180,E1 -4869.262,E2 -4869.262} C_VEL
LIN {X 0,Y 524.013,Z 456.832,A -85,B 0,C 180,E1 -4871.752,E2 -4871.752} C_VEL
LIN {X 0,Y 523.982,Z 456.838,A -85,B 0,C 180,E1 -4875.053,E2 -4875.053} C_VEL
LIN {X 0,Y 523.954,Z 456.839,A -85,B 0,C 180,E1 -4877.97,E2 -4877.97} C_VEL
LIN {X 0,Y 523.962,Z 456.845,A -85,B 0,C 180,E1 -4880.411,E2 -4880.411} C_VEL
LIN {X 0,Y 523.907,Z 456.848,A -85,B 0,C 180,E1 -4882.894,E2 -4882.894} C_VEL
LIN {X 0,Y 523.946,Z 456.839,A -85,B 0,C 180,E1 -4885.419,E2 -4885.419} C_VEL
LIN {X 0,Y 523.962,Z 456.84,A -85,B 0,C 180,E1 -4888,E2 -4888} C_VEL
LIN {X 0,Y 523.944,Z 456.844,A -85,B 0,C 180,E1 -4890.857,E2 -4890.857} C_VEL
LIN {X 0,Y 523.955,Z 456.838,A -85,B 0,C 180,E1 -4893.736,E2 -4893.736} C_VEL
LIN {X 0,Y 523.918,Z 456.852,A -85,B 0,C 180,E1 -4896.406,E2 -4896.406} C_VEL
LIN {X 0,Y 523.953,Z 456.841,A -85,B 0,C 180,E1 -4899.082,E2 -4899.082} C_VEL
LIN {X 0,Y 523.95,Z 456.844,A -85,B 0,C 180,E1 -4902.119,E2 -4902.119} C_VEL
LIN {X 0,Y 523.95,Z 456.84,A -85,B 0,C 180,E1 -4905.31,E2 -4905.31} C_VEL
LIN {X 0,Y 523.917,Z 456.847,A -85,B 0,C 180,E1 -4906.925,E2 -4906.925} C_VEL
LIN {X 0,Y 523.252,Z 456.928,A -85,B 0,C 180,E1 -4907.567,E2 -4907.567} C_VEL
LIN {X 0,Y 520.416,Z 457.288,A -85,B 0,C 180,E1 -4908.609,E2 -4908.609} C_VEL
LIN {X 0,Y 518.02,Z 457.589,A -85,B 0,C 180,E1 -4909.448,E2 -4909.448} C_VEL
LIN {X 0,Y 516.991,Z 457.715,A -85,B 0,C 180,E1 -4910.096,E2 -4910.096} C_VEL
LIN {X 0,Y 516.907,Z 457.724,A -85,B 0,C 180,E1 -4910.315,E2 -4910.315} C_VEL
LIN {X 0,Y 516.881,Z 457.719,A -85,B 0,C 180,E1 -4913.343,E2 -4913.343} C_VEL
LIN {X 0,Y 516.911,Z 457.721,A -85,B 0,C 180,E1 -4916.122,E2 -4916.122} C_VEL
LIN {X 0,Y 516.892,Z 457.723,A -85,B 0,C 180,E1 -4918.936,E2 -4918.936} C_VEL
LIN {X 0,Y 516.923,Z 457.719,A -85,B 0,C 180,E1 -4921.587,E2 -4921.587} C_VEL
LIN {X 0,Y 516.933,Z 457.72,A -85,B 0,C 180,E1 -4924.212,E2 -4924.212} C_VEL
LIN {X 0,Y 516.937,Z 457.799,A -85,B 0,C 180,E1 -4925.146,E2 -4925.146} C_VEL
LIN {X 0,Y 518.846,Z 467.509,A -85,B 0,C 180,E1 -4926.871,E2 -4926.871} C_VEL
LIN {X 0,Y 518.405,Z 482.748,A -85,B 0,C 180,E1 -4929.362,E2 -4929.362} C_VEL
LIN {X 0,Y 517.86,Z 501.781,A -85,B 0,C 180,E1 -4932.428,E2 -4932.428} C_VEL
LIN {X 0,Y 517.495,Z 515.382,A -85,B 0,C 180,E1 -4934.584,E2 -4934.584} C_VEL
LIN {X 0,Y 519.318,Z 526.293,A -85,B 0,C 180,E1 -4934.806,E2 -4934.806} C_VEL
LIN {X 0,Y 518.878,Z 624.35,A -85,B 0,C 180,E1 -4936.165,E2 -4936.165} C_VEL
LIN {X 0,Y 518.671,Z 636.83,A -85,B 0,C 180,E1 -4936.484,E2 -4936.484} C_VEL
LIN {X 0,Y 518.406,Z 649.669,A -85,B 0,C 180,E1 -4936.976,E2 -4936.976} C_VEL
LIN {X 0,Y 518.102,Z 661.639,A -85,B 0,C 180,E1 -4937.601,E2 -4937.601} C_VEL
LIN {X 0,Y 517.826,Z 672.683,A -85,B 0,C 180,E1 -4938.354,E2 -4938.354} C_VEL
LIN {X 0,Y 517.423,Z 683.112,A -85,B 0,C 180,E1 -4939.237,E2 -4939.237} C_VEL
LIN {X 0,Y 517.157,Z 692.515,A -85,B 0,C 180,E1 -4940.221,E2 -4940.221} C_VEL
LIN {X 0,Y 516.865,Z 701.581,A -85,B 0,C 180,E1 -4941.399,E2 -4941.399} C_VEL
LIN {X 0,Y 516.612,Z 708.872,A -85,B 0,C 180,E1 -4942.576,E2 -4942.576} C_VEL
LIN {X 0,Y 516.486,Z 714.725,A -85,B 0,C 180,E1 -4943.752,E2 -4943.752} C_VEL
LIN {X 0,Y 516.321,Z 719.362,A -85,B 0,C 180,E1 -4944.925,E2 -4944.925} C_VEL
LIN {X 0,Y 516.372,Z 722.905,A -85,B 0,C 180,E1 -4946.099,E2 -4946.099} C_VEL
LIN {X 0,Y 516.312,Z 724.743,A -85,B 0,C 180,E1 -4946.88,E2 -4946.88} C_VEL
LIN {X 0,Y 516.261,Z 726.129,A -85,B 0,C 180,E1 -4947.66,E2 -4947.66} C_VEL
LIN {X 0,Y 516.163,Z 727.727,A -85,B 0,C 180,E1 -4949.221,E2 -4949.221} C_VEL
LIN {X 0,Y 516.159,Z 727.96,A -85,B 0,C 180,E1 -4950.001,E2 -4950.001} C_VEL
LIN {X 0,Y 516.163,Z 727.779,A -85,B 0,C 180,E1 -4950.781,E2 -4950.781} C_VEL
LIN {X 0,Y 516.262,Z 726.249,A -85,B 0,C 180,E1 -4952.342,E2 -4952.342} C_VEL
LIN {X 0,Y 516.313,Z 724.913,A -85,B 0,C 180,E1 -4953.122,E2 -4953.122} C_VEL
LIN {X 0,Y 516.362,Z 722.093,A -85,B 0,C 180,E1 -4954.294,E2 -4954.294} C_VEL
LIN {X 0,Y 516.404,Z 718.273,A -85,B 0,C 180,E1 -4955.468,E2 -4955.468} C_VEL
LIN {X 0,Y 516.526,Z 712.484,A -85,B 0,C 180,E1 -4956.823,E2 -4956.823} C_VEL
LIN {X 0,Y 516.731,Z 705.959,A -85,B 0,C 180,E1 -4958.015,E2 -4958.015} C_VEL
LIN {X 0,Y 516.958,Z 697.961,A -85,B 0,C 180,E1 -4959.193,E2 -4959.193} C_VEL
LIN {X 0,Y 517.196,Z 689.793,A -85,B 0,C 180,E1 -4960.176,E2 -4960.176} C_VEL
LIN {X 0,Y 517.559,Z 679.781,A -85,B 0,C 180,E1 -4961.158,E2 -4961.158} C_VEL
LIN {X 0,Y 517.955,Z 668.834,A -85,B 0,C 180,E1 -4962.016,E2 -4962.016} C_VEL
LIN {X 0,Y 518.214,Z 657.351,A -85,B 0,C 180,E1 -4962.732,E2 -4962.732} C_VEL
LIN {X 0,Y 518.525,Z 644.806,A -85,B 0,C 180,E1 -4963.322,E2 -4963.322} C_VEL
LIN {X 0,Y 518.783,Z 632.226,A -85,B 0,C 180,E1 -4963.74,E2 -4963.74} C_VEL
LIN {X 0,Y 518.95,Z 619.261,A -85,B 0,C 180,E1 -4964.01,E2 -4964.01} C_VEL
LIN {X 0,Y 519.231,Z 525.502,A -85,B 0,C 180,E1 -4965.292,E2 -4965.292} C_VEL
LIN {X 0,Y 517.507,Z 515.322,A -85,B 0,C 180,E1 -4965.515,E2 -4965.515} C_VEL
LIN {X 0,Y 518.048,Z 494.838,A -85,B 0,C 180,E1 -4968.776,E2 -4968.776} C_VEL
LIN {X 0,Y 518.645,Z 475.654,A -85,B 0,C 180,E1 -4971.88,E2 -4971.88} C_VEL
LIN {X 0,Y 518.776,Z 466.759,A -85,B 0,C 180,E1 -4973.345,E2 -4973.345} C_VEL
LIN {X 0,Y 516.94,Z 457.721,A -85,B 0,C 180,E1 -4974.981,E2 -4974.981} C_VEL
LIN {X 0,Y 516.933,Z 457.724,A -85,B 0,C 180,E1 -4977.906,E2 -4977.906} C_VEL
LIN {X 0,Y 516.899,Z 457.725,A -85,B 0,C 180,E1 -4980.204,E2 -4980.204} C_VEL
LIN {X 0,Y 516.901,Z 457.72,A -85,B 0,C 180,E1 -4982.947,E2 -4982.947} C_VEL
LIN {X 0,Y 516.877,Z 457.728,A -85,B 0,C 180,E1 -4985.781,E2 -4985.781} C_VEL
LIN {X 0,Y 516.889,Z 457.719,A -85,B 0,C 180,E1 -4988.716,E2 -4988.716} C_VEL
LIN {X 0,Y 516.922,Z 457.723,A -85,B 0,C 180,E1 -4991.775,E2 -4991.775} C_VEL
LIN {X 0,Y 516.929,Z 457.714,A -85,B 0,C 180,E1 -4995.01,E2 -4995.01} C_VEL
LIN {X 0,Y 516.919,Z 457.715,A -85,B 0,C 180,E1 -4998.399,E2 -4998.399} C_VEL
LIN {X 0,Y 516.886,Z 457.723,A -85,B 0,C 180,E1 -5001.284,E2 -5001.284} C_VEL
LIN {X 0,Y 516.897,Z 457.72,A -85,B 0,C 180,E1 -5004.221,E2 -5004.221} C_VEL
LIN {X 0,Y 516.902,Z 457.719,A -85,B 0,C 180,E1 -5007.053,E2 -5007.053} C_VEL
LIN {X 0,Y 516.898,Z 457.726,A -85,B 0,C 180,E1 -5009.796,E2 -5009.796} C_VEL
LIN {X 0,Y 516.932,Z 457.716,A -85,B 0,C 180,E1 -5012.467,E2 -5012.467} C_VEL
LIN {X 0,Y 516.982,Z 457.783,A -85,B 0,C 180,E1 -5014.618,E2 -5014.618} C_VEL
LIN {X 0,Y 518.848,Z 468.069,A -85,B 0,C 180,E1 -5016.235,E2 -5016.235} C_VEL
LIN {X 0,Y 518.369,Z 489.243,A -85,B 0,C 180,E1 -5019.359,E2 -5019.359} C_VEL
LIN {X 0,Y 517.892,Z 510.064,A -85,B 0,C 180,E1 -5022.426,E2 -5022.426} C_VEL
LIN {X 0,Y 517.571,Z 525.429,A -85,B 0,C 180,E1 -5024.693,E2 -5024.693} C_VEL
LIN {X 0,Y 519.086,Z 535.012,A -85,B 0,C 180,E1 -5024.885,E2 -5024.885} C_VEL
LIN {X 0,Y 518.534,Z 633.93,A -85,B 0,C 180,E1 -5026.304,E2 -5026.304} C_VEL
LIN {X 0,Y 518.382,Z 647.322,A -85,B 0,C 180,E1 -5026.65,E2 -5026.65} C_VEL
LIN {X 0,Y 518.134,Z 659.366,A -85,B 0,C 180,E1 -5027.117,E2 -5027.117} C_VEL
LIN {X 0,Y 517.912,Z 670.575,A -85,B 0,C 180,E1 -5027.698,E2 -5027.698} C_VEL
LIN {X 0,Y 517.604,Z 681.891,A -85,B 0,C 180,E1 -5028.447,E2 -5028.447} C_VEL
LIN {X 0,Y 517.293,Z 692.515,A -85,B 0,C 180,E1 -5029.332,E2 -5029.332} C_VEL
LIN {X 0,Y 517.007,Z 702.895,A -85,B 0,C 180,E1 -5030.414,E2 -5030.414} C_VEL
LIN {X 0,Y 516.813,Z 710.558,A -85,B 0,C 180,E1 -5031.397,E2 -5031.397} C_VEL
LIN {X 0,Y 516.573,Z 718.007,A -85,B 0,C 180,E1 -5032.574,E2 -5032.574} C_VEL
LIN {X 0,Y 516.439,Z 723.996,A -85,B 0,C 180,E1 -5033.75,E2 -5033.75} C_VEL
LIN {X 0,Y 516.313,Z 728.738,A -85,B 0,C 180,E1 -5034.924,E2 -5034.924} C_VEL
LIN {X 0,Y 516.373,Z 732.363,A -85,B 0,C 180,E1 -5036.098,E2 -5036.098} C_VEL
LIN {X 0,Y 516.261,Z 735.685,A -85,B 0,C 180,E1 -5037.659,E2 -5037.659} C_VEL
LIN {X 0,Y 516.161,Z 737.292,A -85,B 0,C 180,E1 -5039.22,E2 -5039.22} C_VEL
LIN {X 0,Y 516.155,Z 737.544,A -85,B 0,C 180,E1 -5040,E2 -5040} C_VEL
LIN {X 0,Y 516.192,Z 736.778,A -85,B 0,C 180,E1 -5041.56,E2 -5041.56} C_VEL
LIN {X 0,Y 516.261,Z 735.829,A -85,B 0,C 180,E1 -5042.34,E2 -5042.34} C_VEL
LIN {X 0,Y 516.373,Z 732.631,A -85,B 0,C 180,E1 -5043.902,E2 -5043.902} C_VEL
LIN {X 0,Y 516.313,Z 729.096,A -85,B 0,C 180,E1 -5045.076,E2 -5045.076} C_VEL
LIN {X 0,Y 516.435,Z 724.449,A -85,B 0,C 180,E1 -5046.25,E2 -5046.25} C_VEL
LIN {X 0,Y 516.571,Z 718.558,A -85,B 0,C 180,E1 -5047.426,E2 -5047.426} C_VEL
LIN {X 0,Y 516.792,Z 711.228,A -85,B 0,C 180,E1 -5048.603,E2 -5048.603} C_VEL
LIN {X 0,Y 516.944,Z 703.722,A -85,B 0,C 180,E1 -5049.587,E2 -5049.587} C_VEL
LIN {X 0,Y 517.261,Z 693.497,A -85,B 0,C 180,E1 -5050.668,E2 -5050.668} C_VEL
LIN {X 0,Y 517.574,Z 683.115,A -85,B 0,C 180,E1 -5051.554,E2 -5051.554} C_VEL
LIN {X 0,Y 517.866,Z 671.524,A -85,B 0,C 180,E1 -5052.334,E2 -5052.334} C_VEL
LIN {X 0,Y 518.104,Z 659.051,A -85,B 0,C 180,E1 -5052.983,E2 -5052.983} C_VEL
LIN {X 0,Y 518.338,Z 646.695,A -85,B 0,C 180,E1 -5053.451,E2 -5053.451} C_VEL
LIN {X 0,Y 518.543,Z 632.808,A -85,B 0,C 180,E1 -5053.795,E2 -5053.795} C_VEL
LIN {X 0,Y 518.982,Z 534.292,A -85,B 0,C 180,E1 -5055.221,E2 -5055.221} C_VEL
LIN {X 0,Y 517.578,Z 525.614,A -85,B 0,C 180,E1 -5055.412,E2 -5055.412} C_VEL
LIN {X 0,Y 517.975,Z 506.405,A -85,B 0,C 180,E1 -5058.235,E2 -5058.235} C_VEL
LIN {X 0,Y 518.369,Z 485.192,A -85,B 0,C 180,E1 -5061.264,E2 -5061.264} C_VEL
LIN {X 0,Y 518.599,Z 467.246,A -85,B 0,C 180,E1 -5063.776,E2 -5063.776} C_VEL
LIN {X 0,Y 516.964,Z 457.716,A -85,B 0,C 180,E1 -5065.194,E2 -5065.194} C_VEL
LIN {X 0,Y 516.924,Z 457.724,A -85,B 0,C 180,E1 -5068.415,E2 -5068.415} C_VEL
LIN {X 0,Y 516.894,Z 457.723,A -85,B 0,C 180,E1 -5071.109,E2 -5071.109} C_VEL
LIN {X 0,Y 516.918,Z 457.724,A -85,B 0,C 180,E1 -5073.967,E2 -5073.967} C_VEL
LIN {X 0,Y 516.888,Z 457.722,A -85,B 0,C 180,E1 -5076.745,E2 -5076.745} C_VEL
LIN {X 0,Y 516.887,Z 457.726,A -85,B 0,C 180,E1 -5079.721,E2 -5079.721} C_VEL
LIN {X 0,Y 516.916,Z 457.723,A -85,B 0,C 180,E1 -5081.775,E2 -5081.775} C_VEL
LIN {X 0,Y 516.899,Z 457.72,A -85,B 0,C 180,E1 -5085.007,E2 -5085.007} C_VEL
LIN {X 0,Y 516.919,Z 457.717,A -85,B 0,C 180,E1 -5088.398,E2 -5088.398} C_VEL
LIN {X 0,Y 516.885,Z 457.723,A -85,B 0,C 180,E1 -5091.284,E2 -5091.284} C_VEL
LIN {X 0,Y 516.875,Z 457.724,A -85,B 0,C 180,E1 -5094.219,E2 -5094.219} C_VEL
LIN {X 0,Y 516.899,Z 457.723,A -85,B 0,C 180,E1 -5097.052,E2 -5097.052} C_VEL
LIN {X 0,Y 516.897,Z 457.725,A -85,B 0,C 180,E1 -5099.796,E2 -5099.796} C_VEL
LIN {X 0,Y 516.926,Z 457.722,A -85,B 0,C 180,E1 -5102.905,E2 -5102.905} C_VEL
LIN {X 0,Y 516.969,Z 457.75,A -85,B 0,C 180,E1 -5103.262,E2 -5103.262} C_VEL
LIN {X 0,Y 520.027,Z 471.096,A -85,B 0,C 180,E1 -5105.111,E2 -5105.111} C_VEL
LIN {X 0,Y 519.357,Z 492.393,A -85,B 0,C 180,E1 -5107.734,E2 -5107.734} C_VEL
LIN {X 0,Y 518.555,Z 517.967,A -85,B 0,C 180,E1 -5110.812,E2 -5110.812} C_VEL
LIN {X 0,Y 518.419,Z 523.23,A -85,B 0,C 180,E1 -5111.447,E2 -5111.447} C_VEL
LIN {X 0,Y 520.249,Z 535.666,A -85,B 0,C 180,E1 -5111.698,E2 -5111.698} C_VEL
LIN {X 0,Y 519.448,Z 661.736,A -85,B 0,C 180,E1 -5113.493,E2 -5113.493} C_VEL
LIN {X 0,Y 519.193,Z 676.17,A -85,B 0,C 180,E1 -5113.854,E2 -5113.854} C_VEL
LIN {X 0,Y 518.913,Z 690.497,A -85,B 0,C 180,E1 -5114.384,E2 -5114.384} C_VEL
LIN {X 0,Y 518.588,Z 702.68,A -85,B 0,C 180,E1 -5114.977,E2 -5114.977} C_VEL
LIN {X 0,Y 518.159,Z 715.538,A -85,B 0,C 180,E1 -5115.768,E2 -5115.768} C_VEL
LIN {X 0,Y 517.812,Z 727.247,A -85,B 0,C 180,E1 -5116.659,E2 -5116.659} C_VEL
LIN {X 0,Y 517.438,Z 737.905,A -85,B 0,C 180,E1 -5117.64,E2 -5117.64} C_VEL
LIN {X 0,Y 517.125,Z 748.615,A -85,B 0,C 180,E1 -5118.832,E2 -5118.832} C_VEL
LIN {X 0,Y 516.804,Z 757.377,A -85,B 0,C 180,E1 -5120.014,E2 -5120.014} C_VEL
LIN {X 0,Y 516.607,Z 765.768,A -85,B 0,C 180,E1 -5121.393,E2 -5121.393} C_VEL
LIN {X 0,Y 516.45,Z 771.617,A -85,B 0,C 180,E1 -5122.571,E2 -5122.571} C_VEL
LIN {X 0,Y 516.373,Z 776.415,A -85,B 0,C 180,E1 -5123.748,E2 -5123.748} C_VEL
LIN {X 0,Y 516.306,Z 780.295,A -85,B 0,C 180,E1 -5124.923,E2 -5124.923} C_VEL
LIN {X 0,Y 516.325,Z 783.283,A -85,B 0,C 180,E1 -5126.097,E2 -5126.097} C_VEL
LIN {X 0,Y 516.258,Z 785.995,A -85,B 0,C 180,E1 -5127.658,E2 -5127.658} C_VEL
LIN {X 0,Y 516.157,Z 787.332,A -85,B 0,C 180,E1 -5129.219,E2 -5129.219} C_VEL
LIN {X 0,Y 516.155,Z 787.334,A -85,B 0,C 180,E1 -5130.779,E2 -5130.779} C_VEL
LIN {X 0,Y 516.258,Z 786.001,A -85,B 0,C 180,E1 -5132.34,E2 -5132.34} C_VEL
LIN {X 0,Y 516.324,Z 783.292,A -85,B 0,C 180,E1 -5133.901,E2 -5133.901} C_VEL
LIN {X 0,Y 516.387,Z 779.105,A -85,B 0,C 180,E1 -5135.466,E2 -5135.466} C_VEL
LIN {X 0,Y 516.402,Z 773.324,A -85,B 0,C 180,E1 -5137.035,E2 -5137.035} C_VEL
LIN {X 0,Y 516.598,Z 766.808,A -85,B 0,C 180,E1 -5138.408,E2 -5138.408} C_VEL
LIN {X 0,Y 516.801,Z 758.697,A -85,B 0,C 180,E1 -5139.786,E2 -5139.786} C_VEL
LIN {X 0,Y 517.064,Z 750.2,A -85,B 0,C 180,E1 -5140.969,E2 -5140.969} C_VEL
LIN {X 0,Y 517.405,Z 739.6,A -85,B 0,C 180,E1 -5142.19,E2 -5142.19} C_VEL
LIN {X 0,Y 517.758,Z 728.465,A -85,B 0,C 180,E1 -5143.241,E2 -5143.241} C_VEL
LIN {X 0,Y 518.12,Z 717.021,A -85,B 0,C 180,E1 -5144.131,E2 -5144.131} C_VEL
LIN {X 0,Y 518.531,Z 704.508,A -85,B 0,C 180,E1 -5144.922,E2 -5144.922} C_VEL
LIN {X 0,Y 518.875,Z 691.673,A -85,B 0,C 180,E1 -5145.565,E2 -5145.565} C_VEL
LIN {X 0,Y 519.19,Z 677.45,A -85,B 0,C 180,E1 -5146.103,E2 -5146.103} C_VEL
LIN {X 0,Y 519.426,Z 662.799,A -85,B 0,C 180,E1 -5146.485,E2 -5146.485} C_VEL
LIN {X 0,Y 519.788,Z 618.758,A -85,B 0,C 180,E1 -5147.126,E2 -5147.126} C_VEL
LIN {X 0,Y 520.173,Z 534.465,A -85,B 0,C 180,E1 -5148.322,E2 -5148.322} C_VEL
LIN {X 0,Y 518.407,Z 523.182,A -85,B 0,C 180,E1 -5148.556,E2 -5148.556} C_VEL
LIN {X 0,Y 519.22,Z 495.799,A -85,B 0,C 180,E1 -5151.852,E2 -5151.852} C_VEL
LIN {X 0,Y 520.047,Z 472.027,A -85,B 0,C 180,E1 -5154.766,E2 -5154.766} C_VEL
LIN {X 0,Y 519.09,Z 466.708,A -85,B 0,C 180,E1 -5155.486,E2 -5155.486} C_VEL
LIN {X 0,Y 516.944,Z 457.721,A -85,B 0,C 180,E1 -5156.764,E2 -5156.764} C_VEL
LIN {X 0,Y 516.921,Z 457.717,A -85,B 0,C 180,E1 -5159.525,E2 -5159.525} C_VEL
LIN {X 0,Y 516.897,Z 457.727,A -85,B 0,C 180,E1 -5162.543,E2 -5162.543} C_VEL
LIN {X 0,Y 516.879,Z 457.718,A -85,B 0,C 180,E1 -5165.331,E2 -5165.331} C_VEL
LIN {X 0,Y 516.877,Z 457.722,A -85,B 0,C 180,E1 -5167.942,E2 -5167.942} C_VEL
LIN {X 0,Y 516.902,Z 457.726,A -85,B 0,C 180,E1 -5170.738,E2 -5170.738} C_VEL
LIN {X 0,Y 516.876,Z 457.721,A -85,B 0,C 180,E1 -5173.902,E2 -5173.902} C_VEL
LIN {X 0,Y 516.874,Z 457.722,A -85,B 0,C 180,E1 -5176.106,E2 -5176.106} C_VEL
LIN {X 0,Y 516.896,Z 457.719,A -85,B 0,C 180,E1 -5179.26,E2 -5179.26} C_VEL
LIN {X 0,Y 516.873,Z 457.721,A -85,B 0,C 180,E1 -5182.056,E2 -5182.056} C_VEL
LIN {X 0,Y 516.888,Z 457.718,A -85,B 0,C 180,E1 -5185.176,E2 -5185.176} C_VEL
LIN {X 0,Y 516.874,Z 457.721,A -85,B 0,C 180,E1 -5187.975,E2 -5187.975} C_VEL
LIN {X 0,Y 516.926,Z 457.722,A -85,B 0,C 180,E1 -5190.696,E2 -5190.696} C_VEL
LIN {X 0,Y 516.934,Z 457.714,A -85,B 0,C 180,E1 -5193.803,E2 -5193.803} C_VEL
LIN {X 0,Y 516.862,Z 457.72,A -85,B 0,C 180,E1 -5196.776,E2 -5196.776} C_VEL
LIN {X 0,Y 516.928,Z 457.71,A -85,B 0,C 180,E1 -5199.731,E2 -5199.731} C_VEL
LIN {X 0,Y 516.92,Z 457.724,A -85,B 0,C 180,E1 -5202.596,E2 -5202.596} C_VEL
LIN {X 0,Y 516.93,Z 457.717,A -85,B 0,C 180,E1 -5205.03,E2 -5205.03} C_VEL
LIN {X 0,Y 516.992,Z 457.709,A -85,B 0,C 180,E1 -5208.234,E2 -5208.234} C_VEL
LIN {X 0,Y 516.962,Z 457.71,A -85,B 0,C 180,E1 -5211.4,E2 -5211.4} C_VEL
LIN {X 0,Y 517.035,Z 457.706,A -85,B 0,C 180,E1 -5214.54,E2 -5214.54} C_VEL
LIN {X 0,Y 517.074,Z 457.695,A -85,B 0,C 180,E1 -5217.663,E2 -5217.663} C_VEL
LIN {X 0,Y 517.086,Z 457.701,A -85,B 0,C 180,E1 -5220.779,E2 -5220.779} C_VEL
LIN {X 0,Y 517.007,Z 457.703,A -85,B 0,C 180,E1 -5223.117,E2 -5223.117} C_VEL
LIN {X 0,Y 517,Z 457.71,A -85,B 0,C 180,E1 -5226.243,E2 -5226.243} C_VEL
LIN {X 0,Y 516.947,Z 457.711,A -85,B 0,C 180,E1 -5229.389,E2 -5229.389} C_VEL
LIN {X 0,Y 516.972,Z 457.709,A -85,B 0,C 180,E1 -5231.825,E2 -5231.825} C_VEL
LIN {X 0,Y 516.935,Z 457.715,A -85,B 0,C 180,E1 -5235.148,E2 -5235.148} C_VEL
LIN {X 0,Y 516.916,Z 457.718,A -85,B 0,C 180,E1 -5238.223,E2 -5238.223} C_VEL
LIN {X 0,Y 516.903,Z 457.723,A -85,B 0,C 180,E1 -5240.702,E2 -5240.702} C_VEL
LIN {X 0,Y 516.901,Z 457.72,A -85,B 0,C 180,E1 -5244.073,E2 -5244.073} C_VEL
LIN {X 0,Y 516.92,Z 457.722,A -85,B 0,C 180,E1 -5246.658,E2 -5246.658} C_VEL
LIN {X 0,Y 516.916,Z 457.715,A -85,B 0,C 180,E1 -5249.528,E2 -5249.528} C_VEL
LIN {X 0,Y 516.893,Z 457.726,A -85,B 0,C 180,E1 -5252.545,E2 -5252.545} C_VEL
LIN {X 0,Y 516.876,Z 457.721,A -85,B 0,C 180,E1 -5255.334,E2 -5255.334} C_VEL
LIN {X 0,Y 516.875,Z 457.722,A -85,B 0,C 180,E1 -5257.945,E2 -5257.945} C_VEL
LIN {X 0,Y 516.897,Z 457.724,A -85,B 0,C 180,E1 -5260.741,E2 -5260.741} C_VEL
LIN {X 0,Y 516.876,Z 457.723,A -85,B 0,C 180,E1 -5263.904,E2 -5263.904} C_VEL
LIN {X 0,Y 516.877,Z 457.725,A -85,B 0,C 180,E1 -5266.108,E2 -5266.108} C_VEL
LIN {X 0,Y 516.899,Z 457.719,A -85,B 0,C 180,E1 -5269.262,E2 -5269.262} C_VEL
LIN {X 0,Y 516.907,Z 457.724,A -85,B 0,C 180,E1 -5270.315,E2 -5270.315} C_VEL
LIN {X 0,Y 516.238,Z 457.805,A -85,B 0,C 180,E1 -5270.965,E2 -5270.965} C_VEL
LIN {X 0,Y 513.381,Z 458.16,A -85,B 0,C 180,E1 -5272.02,E2 -5272.02} C_VEL
LIN {X 0,Y 510.961,Z 458.459,A -85,B 0,C 180,E1 -5272.87,E2 -5272.87} C_VEL
LIN {X 0,Y 509.916,Z 458.587,A -85,B 0,C 180,E1 -5273.527,E2 -5273.527} C_VEL
LIN {X 0,Y 509.827,Z 458.598,A -85,B 0,C 180,E1 -5273.749,E2 -5273.749} C_VEL
LIN {X 0,Y 509.861,Z 458.6,A -85,B 0,C 180,E1 -5276.541,E2 -5276.541} C_VEL
LIN {X 0,Y 509.849,Z 458.599,A -85,B 0,C 180,E1 -5279.336,E2 -5279.336} C_VEL
LIN {X 0,Y 509.894,Z 458.598,A -85,B 0,C 180,E1 -5282.056,E2 -5282.056} C_VEL
LIN {X 0,Y 509.926,Z 458.736,A -85,B 0,C 180,E1 -5284.921,E2 -5284.921} C_VEL
LIN {X 0,Y 511.993,Z 469.643,A -85,B 0,C 180,E1 -5286.882,E2 -5286.882} C_VEL
LIN {X 0,Y 511.408,Z 486.802,A -85,B 0,C 180,E1 -5289.715,E2 -5289.715} C_VEL
LIN {X 0,Y 510.85,Z 504.526,A -85,B 0,C 180,E1 -5292.59,E2 -5292.59} C_VEL
LIN {X 0,Y 510.57,Z 515.558,A -85,B 0,C 180,E1 -5294.36,E2 -5294.36} C_VEL
LIN {X 0,Y 512.53,Z 526.735,A -85,B 0,C 180,E1 -5294.582,E2 -5294.582} C_VEL
LIN {X 0,Y 512.084,Z 625.122,A -85,B 0,C 180,E1 -5295.952,E2 -5295.952} C_VEL
LIN {X 0,Y 511.882,Z 638.247,A -85,B 0,C 180,E1 -5296.301,E2 -5296.301} C_VEL
LIN {X 0,Y 511.576,Z 650.833,A -85,B 0,C 180,E1 -5296.799,E2 -5296.799} C_VEL
LIN {X 0,Y 511.234,Z 662.623,A -85,B 0,C 180,E1 -5297.435,E2 -5297.435} C_VEL
LIN {X 0,Y 510.865,Z 674.784,A -85,B 0,C 180,E1 -5298.294,E2 -5298.294} C_VEL
LIN {X 0,Y 510.45,Z 684.905,A -85,B 0,C 180,E1 -5299.189,E2 -5299.189} C_VEL
LIN {X 0,Y 510.197,Z 693.18,A -85,B 0,C 180,E1 -5300.086,E2 -5300.086} C_VEL
LIN {X 0,Y 509.881,Z 702.165,A -85,B 0,C 180,E1 -5301.28,E2 -5301.28} C_VEL
LIN {X 0,Y 509.61,Z 709.407,A -85,B 0,C 180,E1 -5302.473,E2 -5302.473} C_VEL
LIN {X 0,Y 509.447,Z 715.221,A -85,B 0,C 180,E1 -5303.665,E2 -5303.665} C_VEL
LIN {X 0,Y 509.26,Z 719.828,A -85,B 0,C 180,E1 -5304.855,E2 -5304.855} C_VEL
LIN {X 0,Y 509.303,Z 723.346,A -85,B 0,C 180,E1 -5306.045,E2 -5306.045} C_VEL
LIN {X 0,Y 509.259,Z 725.172,A -85,B 0,C 180,E1 -5306.837,E2 -5306.837} C_VEL
LIN {X 0,Y 509.191,Z 726.549,A -85,B 0,C 180,E1 -5307.628,E2 -5307.628} C_VEL
LIN {X 0,Y 509.076,Z 728.138,A -85,B 0,C 180,E1 -5309.21,E2 -5309.21} C_VEL
LIN {X 0,Y 509.072,Z 728.369,A -85,B 0,C 180,E1 -5310.001,E2 -5310.001} C_VEL
LIN {X 0,Y 509.113,Z 727.617,A -85,B 0,C 180,E1 -5311.583,E2 -5311.583} C_VEL
LIN {X 0,Y 509.26,Z 725.337,A -85,B 0,C 180,E1 -5313.165,E2 -5313.165} C_VEL
LIN {X 0,Y 509.29,Z 722.535,A -85,B 0,C 180,E1 -5314.354,E2 -5314.354} C_VEL
LIN {X 0,Y 509.347,Z 718.738,A -85,B 0,C 180,E1 -5315.544,E2 -5315.544} C_VEL
LIN {X 0,Y 509.482,Z 713.134,A -85,B 0,C 180,E1 -5316.889,E2 -5316.889} C_VEL
LIN {X 0,Y 509.732,Z 706.508,A -85,B 0,C 180,E1 -5318.125,E2 -5318.125} C_VEL
LIN {X 0,Y 509.987,Z 698.56,A -85,B 0,C 180,E1 -5319.32,E2 -5319.32} C_VEL
LIN {X 0,Y 510.245,Z 690.455,A -85,B 0,C 180,E1 -5320.316,E2 -5320.316} C_VEL
LIN {X 0,Y 510.646,Z 680.546,A -85,B 0,C 180,E1 -5321.311,E2 -5321.311} C_VEL
LIN {X 0,Y 511.075,Z 669.732,A -85,B 0,C 180,E1 -5322.177,E2 -5322.177} C_VEL
LIN {X 0,Y 511.359,Z 658.323,A -85,B 0,C 180,E1 -5322.906,E2 -5322.906} C_VEL
LIN {X 0,Y 511.717,Z 646.04,A -85,B 0,C 180,E1 -5323.503,E2 -5323.503} C_VEL
LIN {X 0,Y 511.966,Z 633.815,A -85,B 0,C 180,E1 -5323.926,E2 -5323.926} C_VEL
LIN {X 0,Y 512.149,Z 620.074,A -85,B 0,C 180,E1 -5324.225,E2 -5324.225} C_VEL
LIN {X 0,Y 512.401,Z 525.984,A -85,B 0,C 180,E1 -5325.519,E2 -5325.519} C_VEL
LIN {X 0,Y 510.521,Z 515.473,A -85,B 0,C 180,E1 -5325.742,E2 -5325.742} C_VEL
LIN {X 0,Y 511.113,Z 496.113,A -85,B 0,C 180,E1 -5328.853,E2 -5328.853} C_VEL
LIN {X 0,Y 511.74,Z 477.055,A -85,B 0,C 180,E1 -5331.978,E2 -5331.978} C_VEL
LIN {X 0,Y 512.021,Z 470.124,A -85,B 0,C 180,E1 -5333.126,E2 -5333.126} C_VEL
LIN {X 0,Y 510.497,Z 461.393,A -85,B 0,C 180,E1 -5334.684,E2 -5334.684} C_VEL
LIN {X 0,Y 509.872,Z 458.602,A -85,B 0,C 180,E1 -5335.206,E2 -5335.206} C_VEL
LIN {X 0,Y 509.904,Z 458.598,A -85,B 0,C 180,E1 -5338.101,E2 -5338.101} C_VEL
LIN {X 0,Y 509.852,Z 458.605,A -85,B 0,C 180,E1 -5341.28,E2 -5341.28} C_VEL
LIN {X 0,Y 509.862,Z 458.597,A -85,B 0,C 180,E1 -5344.203,E2 -5344.203} C_VEL
LIN {X 0,Y 509.823,Z 458.604,A -85,B 0,C 180,E1 -5347.341,E2 -5347.341} C_VEL
LIN {X 0,Y 509.845,Z 458.598,A -85,B 0,C 180,E1 -5350.382,E2 -5350.382} C_VEL
LIN {X 0,Y 509.847,Z 458.599,A -85,B 0,C 180,E1 -5353.065,E2 -5353.065} C_VEL
LIN {X 0,Y 509.837,Z 458.606,A -85,B 0,C 180,E1 -5355.793,E2 -5355.793} C_VEL
LIN {X 0,Y 509.861,Z 458.594,A -85,B 0,C 180,E1 -5358.575,E2 -5358.575} C_VEL
LIN {X 0,Y 509.857,Z 458.598,A -85,B 0,C 180,E1 -5361.787,E2 -5361.787} C_VEL
LIN {X 0,Y 509.852,Z 458.596,A -85,B 0,C 180,E1 -5364.623,E2 -5364.623} C_VEL
LIN {X 0,Y 509.869,Z 458.6,A -85,B 0,C 180,E1 -5367.481,E2 -5367.481} C_VEL
LIN {X 0,Y 509.864,Z 458.598,A -85,B 0,C 180,E1 -5370.274,E2 -5370.274} C_VEL
LIN {X 0,Y 509.889,Z 458.594,A -85,B 0,C 180,E1 -5372.944,E2 -5372.944} C_VEL
LIN {X 0,Y 509.948,Z 458.722,A -85,B 0,C 180,E1 -5374.434,E2 -5374.434} C_VEL
LIN {X 0,Y 511.942,Z 469.312,A -85,B 0,C 180,E1 -5376.11,E2 -5376.11} C_VEL
LIN {X 0,Y 511.479,Z 489.176,A -85,B 0,C 180,E1 -5379.068,E2 -5379.068} C_VEL
LIN {X 0,Y 510.923,Z 511.543,A -85,B 0,C 180,E1 -5382.385,E2 -5382.385} C_VEL
LIN {X 0,Y 510.612,Z 525.705,A -85,B 0,C 180,E1 -5384.481,E2 -5384.481} C_VEL
LIN {X 0,Y 512.24,Z 536.279,A -85,B 0,C 180,E1 -5384.696,E2 -5384.696} C_VEL
LIN {X 0,Y 511.62,Z 634.506,A -85,B 0,C 180,E1 -5386.141,E2 -5386.141} C_VEL
LIN {X 0,Y 511.443,Z 647.76,A -85,B 0,C 180,E1 -5386.49,E2 -5386.49} C_VEL
LIN {X 0,Y 511.182,Z 660.278,A -85,B 0,C 180,E1 -5386.989,E2 -5386.989} C_VEL
LIN {X 0,Y 510.942,Z 671.458,A -85,B 0,C 180,E1 -5387.584,E2 -5387.584} C_VEL
LIN {X 0,Y 510.593,Z 683.253,A -85,B 0,C 180,E1 -5388.387,E2 -5388.387} C_VEL
LIN {X 0,Y 510.28,Z 693.635,A -85,B 0,C 180,E1 -5389.284,E2 -5389.284} C_VEL
LIN {X 0,Y 509.985,Z 703.024,A -85,B 0,C 180,E1 -5390.281,E2 -5390.281} C_VEL
LIN {X 0,Y 509.771,Z 710.736,A -85,B 0,C 180,E1 -5391.277,E2 -5391.277} C_VEL
LIN {X 0,Y 509.531,Z 718.259,A -85,B 0,C 180,E1 -5392.471,E2 -5392.471} C_VEL
LIN {X 0,Y 509.389,Z 724.273,A -85,B 0,C 180,E1 -5393.663,E2 -5393.663} C_VEL
LIN {X 0,Y 509.248,Z 729.032,A -85,B 0,C 180,E1 -5394.853,E2 -5394.853} C_VEL
LIN {X 0,Y 509.304,Z 732.671,A -85,B 0,C 180,E1 -5396.044,E2 -5396.044} C_VEL
LIN {X 0,Y 509.202,Z 734.553,A -85,B 0,C 180,E1 -5396.835,E2 -5396.835} C_VEL
LIN {X 0,Y 509.19,Z 735.994,A -85,B 0,C 180,E1 -5397.627,E2 -5397.627} C_VEL
LIN {X 0,Y 509.075,Z 737.631,A -85,B 0,C 180,E1 -5399.209,E2 -5399.209} C_VEL
LIN {X 0,Y 509.066,Z 737.875,A -85,B 0,C 180,E1 -5400,E2 -5400} C_VEL
LIN {X 0,Y 509.075,Z 737.694,A -85,B 0,C 180,E1 -5400.791,E2 -5400.791} C_VEL
LIN {X 0,Y 509.19,Z 736.149,A -85,B 0,C 180,E1 -5402.373,E2 -5402.373} C_VEL
LIN {X 0,Y 509.202,Z 734.783,A -85,B 0,C 180,E1 -5403.165,E2 -5403.165} C_VEL
LIN {X 0,Y 509.284,Z 731.914,A -85,B 0,C 180,E1 -5404.353,E2 -5404.353} C_VEL
LIN {X 0,Y 509.345,Z 728.007,A -85,B 0,C 180,E1 -5405.543,E2 -5405.543} C_VEL
LIN {X 0,Y 509.421,Z 722.295,A -85,B 0,C 180,E1 -5406.864,E2 -5406.864} C_VEL
LIN {X 0,Y 509.643,Z 715.337,A -85,B 0,C 180,E1 -5408.126,E2 -5408.126} C_VEL
LIN {X 0,Y 509.827,Z 707.066,A -85,B 0,C 180,E1 -5409.321,E2 -5409.321} C_VEL
LIN {X 0,Y 510.098,Z 698.549,A -85,B 0,C 180,E1 -5410.318,E2 -5410.318} C_VEL
LIN {X 0,Y 510.482,Z 688.077,A -85,B 0,C 180,E1 -5411.314,E2 -5411.314} C_VEL
LIN {X 0,Y 510.775,Z 677.007,A -85,B 0,C 180,E1 -5412.151,E2 -5412.151} C_VEL
LIN {X 0,Y 510.995,Z 665.961,A -85,B 0,C 180,E1 -5412.813,E2 -5412.813} C_VEL
LIN {X 0,Y 511.308,Z 654.032,A -85,B 0,C 180,E1 -5413.361,E2 -5413.361} C_VEL
LIN {X 0,Y 511.513,Z 640.901,A -85,B 0,C 180,E1 -5413.786,E2 -5413.786} C_VEL
LIN {X 0,Y 511.675,Z 626.831,A -85,B 0,C 180,E1 -5414.06,E2 -5414.06} C_VEL
LIN {X 0,Y 512.135,Z 535.367,A -85,B 0,C 180,E1 -5415.409,E2 -5415.409} C_VEL
LIN {X 0,Y 510.683,Z 526.051,A -85,B 0,C 180,E1 -5415.618,E2 -5415.618} C_VEL
LIN {X 0,Y 511.093,Z 505.33,A -85,B 0,C 180,E1 -5418.645,E2 -5418.645} C_VEL
LIN {X 0,Y 511.432,Z 487.97,A -85,B 0,C 180,E1 -5421.145,E2 -5421.145} C_VEL
LIN {X 0,Y 511.677,Z 468.448,A -85,B 0,C 180,E1 -5423.903,E2 -5423.903} C_VEL
LIN {X 0,Y 509.912,Z 458.595,A -85,B 0,C 180,E1 -5425.349,E2 -5425.349} C_VEL
LIN {X 0,Y 509.903,Z 458.598,A -85,B 0,C 180,E1 -5428.101,E2 -5428.101} C_VEL
LIN {X 0,Y 509.851,Z 458.6,A -85,B 0,C 180,E1 -5431.28,E2 -5431.28} C_VEL
LIN {X 0,Y 509.866,Z 458.602,A -85,B 0,C 180,E1 -5434.203,E2 -5434.203} C_VEL
LIN {X 0,Y 509.824,Z 458.602,A -85,B 0,C 180,E1 -5437.34,E2 -5437.34} C_VEL
LIN {X 0,Y 509.842,Z 458.602,A -85,B 0,C 180,E1 -5440.382,E2 -5440.382} C_VEL
LIN {X 0,Y 509.827,Z 458.601,A -85,B 0,C 180,E1 -5443.062,E2 -5443.062} C_VEL
LIN {X 0,Y 509.828,Z 458.606,A -85,B 0,C 180,E1 -5445.793,E2 -5445.793} C_VEL
LIN {X 0,Y 509.861,Z 458.596,A -85,B 0,C 180,E1 -5448.574,E2 -5448.574} C_VEL
LIN {X 0,Y 509.855,Z 458.602,A -85,B 0,C 180,E1 -5451.786,E2 -5451.786} C_VEL
LIN {X 0,Y 509.834,Z 458.6,A -85,B 0,C 180,E1 -5454.621,E2 -5454.621} C_VEL
LIN {X 0,Y 509.866,Z 458.602,A -85,B 0,C 180,E1 -5457.48,E2 -5457.48} C_VEL
LIN {X 0,Y 509.863,Z 458.599,A -85,B 0,C 180,E1 -5460.273,E2 -5460.273} C_VEL
LIN {X 0,Y 509.92,Z 458.674,A -85,B 0,C 180,E1 -5463.006,E2 -5463.006} C_VEL
LIN {X 0,Y 513.064,Z 471.87,A -85,B 0,C 180,E1 -5464.871,E2 -5464.871} C_VEL
LIN {X 0,Y 513.057,Z 478.657,A -85,B 0,C 180,E1 -5465.735,E2 -5465.735} C_VEL
LIN {X 0,Y 512.1,Z 503.557,A -85,B 0,C 180,E1 -5468.815,E2 -5468.815} C_VEL
LIN {X 0,Y 511.512,Z 523.237,A -85,B 0,C 180,E1 -5471.219,E2 -5471.219} C_VEL
LIN {X 0,Y 513.46,Z 536.17,A -85,B 0,C 180,E1 -5471.478,E2 -5471.478} C_VEL
LIN {X 0,Y 512.551,Z 662.082,A -85,B 0,C 180,E1 -5473.312,E2 -5473.312} C_VEL
LIN {X 0,Y 512.215,Z 676.763,A -85,B 0,C 180,E1 -5473.694,E2 -5473.694} C_VEL
LIN {X 0,Y 511.981,Z 690.535,A -85,B 0,C 180,E1 -5474.218,E2 -5474.218} C_VEL
LIN {X 0,Y 511.613,Z 703.526,A -85,B 0,C 180,E1 -5474.87,E2 -5474.87} C_VEL
LIN {X 0,Y 511.129,Z 716.151,A -85,B 0,C 180,E1 -5475.67,E2 -5475.67} C_VEL
LIN {X 0,Y 510.766,Z 727.693,A -85,B 0,C 180,E1 -5476.573,E2 -5476.573} C_VEL
LIN {X 0,Y 510.377,Z 738.585,A -85,B 0,C 180,E1 -5477.604,E2 -5477.604} C_VEL
LIN {X 0,Y 510.092,Z 747.995,A -85,B 0,C 180,E1 -5478.676,E2 -5478.676} C_VEL
LIN {X 0,Y 509.763,Z 756.806,A -85,B 0,C 180,E1 -5479.875,E2 -5479.875} C_VEL
LIN {X 0,Y 509.548,Z 765.248,A -85,B 0,C 180,E1 -5481.273,E2 -5481.273} C_VEL
LIN {X 0,Y 509.373,Z 771.121,A -85,B 0,C 180,E1 -5482.467,E2 -5482.467} C_VEL
LIN {X 0,Y 509.288,Z 775.943,A -85,B 0,C 180,E1 -5483.661,E2 -5483.661} C_VEL
LIN {X 0,Y 509.239,Z 779.849,A -85,B 0,C 180,E1 -5484.852,E2 -5484.852} C_VEL
LIN {X 0,Y 509.235,Z 782.848,A -85,B 0,C 180,E1 -5486.042,E2 -5486.042} C_VEL
LIN {X 0,Y 509.187,Z 785.596,A -85,B 0,C 180,E1 -5487.626,E2 -5487.626} C_VEL
LIN {X 0,Y 509.071,Z 786.952,A -85,B 0,C 180,E1 -5489.208,E2 -5489.208} C_VEL
LIN {X 0,Y 509.069,Z 786.953,A -85,B 0,C 180,E1 -5490.79,E2 -5490.79} C_VEL
LIN {X 0,Y 509.187,Z 785.602,A -85,B 0,C 180,E1 -5492.372,E2 -5492.372} C_VEL
LIN {X 0,Y 509.234,Z 782.86,A -85,B 0,C 180,E1 -5493.956,E2 -5493.956} C_VEL
LIN {X 0,Y 509.299,Z 778.651,A -85,B 0,C 180,E1 -5495.542,E2 -5495.542} C_VEL
LIN {X 0,Y 509.327,Z 772.844,A -85,B 0,C 180,E1 -5497.133,E2 -5497.133} C_VEL
LIN {X 0,Y 509.502,Z 766.292,A -85,B 0,C 180,E1 -5498.526,E2 -5498.526} C_VEL
LIN {X 0,Y 509.734,Z 758.14,A -85,B 0,C 180,E1 -5499.923,E2 -5499.923} C_VEL
LIN {X 0,Y 510.017,Z 749.599,A -85,B 0,C 180,E1 -5501.122,E2 -5501.122} C_VEL
LIN {X 0,Y 510.344,Z 739.664,A -85,B 0,C 180,E1 -5502.283,E2 -5502.283} C_VEL
LIN {X 0,Y 510.729,Z 728.901,A -85,B 0,C 180,E1 -5503.325,E2 -5503.325} C_VEL
LIN {X 0,Y 511.112,Z 717.631,A -85,B 0,C 180,E1 -5504.227,E2 -5504.227} C_VEL
LIN {X 0,Y 511.533,Z 705.353,A -85,B 0,C 180,E1 -5505.029,E2 -5505.029} C_VEL
LIN {X 0,Y 511.939,Z 691.713,A -85,B 0,C 180,E1 -5505.73,E2 -5505.73} C_VEL
LIN {X 0,Y 512.268,Z 677.67,A -85,B 0,C 180,E1 -5506.275,E2 -5506.275} C_VEL
LIN {X 0,Y 512.518,Z 663.261,A -85,B 0,C 180,E1 -5506.662,E2 -5506.662} C_VEL
LIN {X 0,Y 512.767,Z 635.811,A -85,B 0,C 180,E1 -5507.086,E2 -5507.086} C_VEL
LIN {X 0,Y 513.429,Z 536.307,A -85,B 0,C 180,E1 -5508.521,E2 -5508.521} C_VEL
LIN {X 0,Y 511.47,Z 523.175,A -85,B 0,C 180,E1 -5508.786,E2 -5508.786} C_VEL
LIN {X 0,Y 512.319,Z 497.324,A -85,B 0,C 180,E1 -5511.95,E2 -5511.95} C_VEL
LIN {X 0,Y 513.186,Z 475.279,A -85,B 0,C 180,E1 -5514.688,E2 -5514.688} C_VEL
LIN {X 0,Y 512.844,Z 471.013,A -85,B 0,C 180,E1 -5515.249,E2 -5515.249} C_VEL
LIN {X 0,Y 509.887,Z 458.599,A -85,B 0,C 180,E1 -5517.014,E2 -5517.014} C_VEL
LIN {X 0,Y 509.877,Z 458.594,A -85,B 0,C 180,E1 -5519.748,E2 -5519.748} C_VEL
LIN {X 0,Y 509.873,Z 458.602,A -85,B 0,C 180,E1 -5522.774,E2 -5522.774} C_VEL
LIN {X 0,Y 509.838,Z 458.594,A -85,B 0,C 180,E1 -5525.58,E2 -5525.58} C_VEL
LIN {X 0,Y 509.853,Z 458.601,A -85,B 0,C 180,E1 -5528.336,E2 -5528.336} C_VEL
LIN {X 0,Y 509.865,Z 458.596,A -85,B 0,C 180,E1 -5531.423,E2 -5531.423} C_VEL
LIN {X 0,Y 509.849,Z 458.605,A -85,B 0,C 180,E1 -5534.667,E2 -5534.667} C_VEL
LIN {X 0,Y 509.855,Z 458.596,A -85,B 0,C 180,E1 -5538.101,E2 -5538.101} C_VEL
LIN {X 0,Y 509.869,Z 458.599,A -85,B 0,C 180,E1 -5540.65,E2 -5540.65} C_VEL
LIN {X 0,Y 509.826,Z 458.592,A -85,B 0,C 180,E1 -5543.647,E2 -5543.647} C_VEL
LIN {X 0,Y 509.854,Z 458.6,A -85,B 0,C 180,E1 -5546.539,E2 -5546.539} C_VEL
LIN {X 0,Y 509.841,Z 458.597,A -85,B 0,C 180,E1 -5549.334,E2 -5549.334} C_VEL
LIN {X 0,Y 509.885,Z 458.592,A -85,B 0,C 180,E1 -5552.054,E2 -5552.054} C_VEL
LIN {X 0,Y 509.868,Z 458.6,A -85,B 0,C 180,E1 -5554.704,E2 -5554.704} C_VEL
LIN {X 0,Y 509.825,Z 458.589,A -85,B 0,C 180,E1 -5557.455,E2 -5557.455} C_VEL
LIN {X 0,Y 509.906,Z 458.585,A -85,B 0,C 180,E1 -5559.844,E2 -5559.844} C_VEL
LIN {X 0,Y 509.877,Z 458.593,A -85,B 0,C 180,E1 -5563.175,E2 -5563.175} C_VEL
LIN {X 0,Y 509.853,Z 458.595,A -85,B 0,C 180,E1 -5565.634,E2 -5565.634} C_VEL
LIN {X 0,Y 509.915,Z 458.591,A -85,B 0,C 180,E1 -5568.875,E2 -5568.875} C_VEL
LIN {X 0,Y 509.941,Z 458.587,A -85,B 0,C 180,E1 -5572.078,E2 -5572.078} C_VEL
LIN {X 0,Y 509.984,Z 458.582,A -85,B 0,C 180,E1 -5574.464,E2 -5574.464} C_VEL
LIN {X 0,Y 510.045,Z 458.57,A -85,B 0,C 180,E1 -5577.631,E2 -5577.631} C_VEL
LIN {X 0,Y 510.056,Z 458.576,A -85,B 0,C 180,E1 -5580.79,E2 -5580.79} C_VEL
LIN {X 0,Y 509.95,Z 458.581,A -85,B 0,C 180,E1 -5583.16,E2 -5583.16} C_VEL
LIN {X 0,Y 509.968,Z 458.587,A -85,B 0,C 180,E1 -5586.33,E2 -5586.33} C_VEL
LIN {X 0,Y 509.908,Z 458.594,A -85,B 0,C 180,E1 -5588.72,E2 -5588.72} C_VEL
LIN {X 0,Y 509.94,Z 458.586,A -85,B 0,C 180,E1 -5591.931,E2 -5591.931} C_VEL
LIN {X 0,Y 509.882,Z 458.593,A -85,B 0,C 180,E1 -5595.242,E2 -5595.242} C_VEL
LIN {X 0,Y 509.878,Z 458.592,A -85,B 0,C 180,E1 -5598.002,E2 -5598.002} C_VEL
LIN {X 0,Y 509.841,Z 458.599,A -85,B 0,C 180,E1 -5601.002,E2 -5601.002} C_VEL
LIN {X 0,Y 509.827,Z 458.599,A -85,B 0,C 180,E1 -5603.564,E2 -5603.564} C_VEL
LIN {X 0,Y 509.904,Z 458.595,A -85,B 0,C 180,E1 -5606.38,E2 -5606.38} C_VEL
LIN {X 0,Y 509.877,Z 458.596,A -85,B 0,C 180,E1 -5608.844,E2 -5608.844} C_VEL
LIN {X 0,Y 509.818,Z 458.6,A -85,B 0,C 180,E1 -5611.591,E2 -5611.591} C_VEL
LIN {X 0,Y 509.847,Z 458.602,A -85,B 0,C 180,E1 -5614.414,E2 -5614.414} C_VEL
LIN {X 0,Y 509.812,Z 458.6,A -85,B 0,C 180,E1 -5617.341,E2 -5617.341} C_VEL
LIN {X 0,Y 509.855,Z 458.602,A -85,B 0,C 180,E1 -5620.381,E2 -5620.381} C_VEL
LIN {X 0,Y 509.817,Z 458.602,A -85,B 0,C 180,E1 -5623.063,E2 -5623.063} C_VEL
LIN {X 0,Y 509.824,Z 458.6,A -85,B 0,C 180,E1 -5625.793,E2 -5625.793} C_VEL
LIN {X 0,Y 509.861,Z 458.603,A -85,B 0,C 180,E1 -5628.577,E2 -5628.577} C_VEL
LIN {X 0,Y 509.855,Z 458.597,A -85,B 0,C 180,E1 -5631.664,E2 -5631.664} C_VEL
LIN {X 0,Y 509.827,Z 458.598,A -85,B 0,C 180,E1 -5633.749,E2 -5633.749} C_VEL
LIN {X 0,Y 509.163,Z 458.689,A -85,B 0,C 180,E1 -5634.409,E2 -5634.409} C_VEL
LIN {X 0,Y 506.344,Z 459.039,A -85,B 0,C 180,E1 -5635.481,E2 -5635.481} C_VEL
LIN {X 0,Y 503.951,Z 459.336,A -85,B 0,C 180,E1 -5636.344,E2 -5636.344} C_VEL
LIN {X 0,Y 502.903,Z 459.466,A -85,B 0,C 180,E1 -5637.011,E2 -5637.011} C_VEL
LIN {X 0,Y 502.806,Z 459.476,A -85,B 0,C 180,E1 -5637.236,E2 -5637.236} C_VEL
LIN {X 0,Y 502.829,Z 459.477,A -85,B 0,C 180,E1 -5640.063,E2 -5640.063} C_VEL
LIN {X 0,Y 502.834,Z 459.476,A -85,B 0,C 180,E1 -5642.535,E2 -5642.535} C_VEL
LIN {X 0,Y 502.863,Z 459.523,A -85,B 0,C 180,E1 -5644.66,E2 -5644.66} C_VEL
LIN {X 0,Y 505.075,Z 470.617,A -85,B 0,C 180,E1 -5646.69,E2 -5646.69} C_VEL
LIN {X 0,Y 504.572,Z 485.994,A -85,B 0,C 180,E1 -5649.269,E2 -5649.269} C_VEL
LIN {X 0,Y 503.916,Z 504.673,A -85,B 0,C 180,E1 -5652.343,E2 -5652.343} C_VEL
LIN {X 0,Y 503.606,Z 515.581,A -85,B 0,C 180,E1 -5654.11,E2 -5654.11} C_VEL
LIN {X 0,Y 505.675,Z 527.14,A -85,B 0,C 180,E1 -5654.349,E2 -5654.349} C_VEL
LIN {X 0,Y 505.308,Z 621.812,A -85,B 0,C 180,E1 -5655.657,E2 -5655.657} C_VEL
LIN {X 0,Y 505.156,Z 635.028,A -85,B 0,C 180,E1 -5655.961,E2 -5655.961} C_VEL
LIN {X 0,Y 504.888,Z 647.522,A -85,B 0,C 180,E1 -5656.416,E2 -5656.416} C_VEL
LIN {X 0,Y 504.537,Z 659.538,A -85,B 0,C 180,E1 -5657.021,E2 -5657.021} C_VEL
LIN {X 0,Y 504.159,Z 670.372,A -85,B 0,C 180,E1 -5657.727,E2 -5657.727} C_VEL
LIN {X 0,Y 503.737,Z 681.444,A -85,B 0,C 180,E1 -5658.636,E2 -5658.636} C_VEL
LIN {X 0,Y 503.4,Z 690.363,A -85,B 0,C 180,E1 -5659.544,E2 -5659.544} C_VEL
LIN {X 0,Y 502.986,Z 699.999,A -85,B 0,C 180,E1 -5660.755,E2 -5660.755} C_VEL
LIN {X 0,Y 502.66,Z 707.754,A -85,B 0,C 180,E1 -5661.964,E2 -5661.964} C_VEL
LIN {X 0,Y 502.409,Z 714.579,A -85,B 0,C 180,E1 -5663.312,E2 -5663.312} C_VEL
LIN {X 0,Y 502.295,Z 718.91,A -85,B 0,C 180,E1 -5664.38,E2 -5664.38} C_VEL
LIN {X 0,Y 502.223,Z 722.759,A -85,B 0,C 180,E1 -5665.587,E2 -5665.587} C_VEL
LIN {X 0,Y 502.207,Z 725.606,A -85,B 0,C 180,E1 -5666.792,E2 -5666.792} C_VEL
LIN {X 0,Y 502.036,Z 727.948,A -85,B 0,C 180,E1 -5668.397,E2 -5668.397} C_VEL
LIN {X 0,Y 501.986,Z 728.778,A -85,B 0,C 180,E1 -5670.001,E2 -5670.001} C_VEL
LIN {X 0,Y 502.037,Z 728.03,A -85,B 0,C 180,E1 -5671.605,E2 -5671.605} C_VEL
LIN {X 0,Y 502.191,Z 725.766,A -85,B 0,C 180,E1 -5673.21,E2 -5673.21} C_VEL
LIN {X 0,Y 502.223,Z 722.984,A -85,B 0,C 180,E1 -5674.415,E2 -5674.415} C_VEL
LIN {X 0,Y 502.292,Z 719.213,A -85,B 0,C 180,E1 -5675.622,E2 -5675.622} C_VEL
LIN {X 0,Y 502.427,Z 714.351,A -85,B 0,C 180,E1 -5676.829,E2 -5676.829} C_VEL
LIN {X 0,Y 502.642,Z 708.247,A -85,B 0,C 180,E1 -5678.038,E2 -5678.038} C_VEL
LIN {X 0,Y 502.95,Z 700.628,A -85,B 0,C 180,E1 -5679.248,E2 -5679.248} C_VEL
LIN {X 0,Y 503.302,Z 691.123,A -85,B 0,C 180,E1 -5680.46,E2 -5680.46} C_VEL
LIN {X 0,Y 503.741,Z 681.297,A -85,B 0,C 180,E1 -5681.468,E2 -5681.468} C_VEL
LIN {X 0,Y 504.201,Z 670.618,A -85,B 0,C 180,E1 -5682.344,E2 -5682.344} C_VEL
LIN {X 0,Y 504.51,Z 659.298,A -85,B 0,C 180,E1 -5683.084,E2 -5683.084} C_VEL
LIN {X 0,Y 504.914,Z 647.21,A -85,B 0,C 180,E1 -5683.688,E2 -5683.688} C_VEL
LIN {X 0,Y 505.176,Z 634.509,A -85,B 0,C 180,E1 -5684.143,E2 -5684.143} C_VEL
LIN {X 0,Y 505.378,Z 620.919,A -85,B 0,C 180,E1 -5684.446,E2 -5684.446} C_VEL
LIN {X 0,Y 505.66,Z 527.02,A -85,B 0,C 180,E1 -5685.743,E2 -5685.743} C_VEL
LIN {X 0,Y 503.6,Z 515.593,A -85,B 0,C 180,E1 -5685.979,E2 -5685.979} C_VEL
LIN {X 0,Y 504.162,Z 496.253,A -85,B 0,C 180,E1 -5689.123,E2 -5689.123} C_VEL
LIN {X 0,Y 504.851,Z 478.455,A -85,B 0,C 180,E1 -5692.079,E2 -5692.079} C_VEL
LIN {X 0,Y 505.016,Z 470.108,A -85,B 0,C 180,E1 -5693.489,E2 -5693.489} C_VEL
LIN {X 0,Y 502.855,Z 459.475,A -85,B 0,C 180,E1 -5695.453,E2 -5695.453} C_VEL
LIN {X 0,Y 502.847,Z 459.476,A -85,B 0,C 180,E1 -5698.373,E2 -5698.373} C_VEL
LIN {X 0,Y 502.799,Z 459.484,A -85,B 0,C 180,E1 -5701.499,E2 -5701.499} C_VEL
LIN {X 0,Y 502.81,Z 459.478,A -85,B 0,C 180,E1 -5703.994,E2 -5703.994} C_VEL
LIN {X 0,Y 502.784,Z 459.479,A -85,B 0,C 180,E1 -5707.178,E2 -5707.178} C_VEL
LIN {X 0,Y 502.795,Z 459.48,A -85,B 0,C 180,E1 -5710.015,E2 -5710.015} C_VEL
LIN {X 0,Y 502.809,Z 459.477,A -85,B 0,C 180,E1 -5712.2,E2 -5712.2} C_VEL
LIN {X 0,Y 502.807,Z 459.478,A -85,B 0,C 180,E1 -5715.468,E2 -5715.468} C_VEL
LIN {X 0,Y 502.825,Z 459.471,A -85,B 0,C 180,E1 -5718.934,E2 -5718.934} C_VEL
LIN {X 0,Y 502.8,Z 459.476,A -85,B 0,C 180,E1 -5722.046,E2 -5722.046} C_VEL
LIN {X 0,Y 502.816,Z 459.474,A -85,B 0,C 180,E1 -5725.035,E2 -5725.035} C_VEL
LIN {X 0,Y 502.791,Z 459.482,A -85,B 0,C 180,E1 -5727.916,E2 -5727.916} C_VEL
LIN {X 0,Y 502.83,Z 459.472,A -85,B 0,C 180,E1 -5730.712,E2 -5730.712} C_VEL
LIN {X 0,Y 502.885,Z 459.471,A -85,B 0,C 180,E1 -5734.104,E2 -5734.104} C_VEL
LIN {X 0,Y 502.893,Z 459.497,A -85,B 0,C 180,E1 -5734.216,E2 -5734.216} C_VEL
LIN {X 0,Y 505.019,Z 470.516,A -85,B 0,C 180,E1 -5735.98,E2 -5735.98} C_VEL
LIN {X 0,Y 504.591,Z 489.16,A -85,B 0,C 180,E1 -5738.769,E2 -5738.769} C_VEL
LIN {X 0,Y 504.036,Z 510.561,A -85,B 0,C 180,E1 -5741.975,E2 -5741.975} C_VEL
LIN {X 0,Y 503.698,Z 525.943,A -85,B 0,C 180,E1 -5744.259,E2 -5744.259} C_VEL
LIN {X 0,Y 505.402,Z 537.379,A -85,B 0,C 180,E1 -5744.499,E2 -5744.499} C_VEL
LIN {X 0,Y 504.7,Z 635.061,A -85,B 0,C 180,E1 -5745.973,E2 -5745.973} C_VEL
LIN {X 0,Y 504.549,Z 647.401,A -85,B 0,C 180,E1 -5746.302,E2 -5746.302} C_VEL
LIN {X 0,Y 504.246,Z 660.133,A -85,B 0,C 180,E1 -5746.807,E2 -5746.807} C_VEL
LIN {X 0,Y 503.937,Z 672.662,A -85,B 0,C 180,E1 -5747.485,E2 -5747.485} C_VEL
LIN {X 0,Y 503.643,Z 683.286,A -85,B 0,C 180,E1 -5748.224,E2 -5748.224} C_VEL
LIN {X 0,Y 503.298,Z 693.725,A -85,B 0,C 180,E1 -5749.134,E2 -5749.134} C_VEL
LIN {X 0,Y 502.982,Z 703.16,A -85,B 0,C 180,E1 -5750.144,E2 -5750.144} C_VEL
LIN {X 0,Y 502.753,Z 710.911,A -85,B 0,C 180,E1 -5751.154,E2 -5751.154} C_VEL
LIN {X 0,Y 502.484,Z 718.478,A -85,B 0,C 180,E1 -5752.364,E2 -5752.364} C_VEL
LIN {X 0,Y 502.326,Z 724.52,A -85,B 0,C 180,E1 -5753.573,E2 -5753.573} C_VEL
LIN {X 0,Y 502.186,Z 729.304,A -85,B 0,C 180,E1 -5754.781,E2 -5754.781} C_VEL
LIN {X 0,Y 502.236,Z 732.964,A -85,B 0,C 180,E1 -5755.988,E2 -5755.988} C_VEL
LIN {X 0,Y 502.125,Z 734.854,A -85,B 0,C 180,E1 -5756.79,E2 -5756.79} C_VEL
LIN {X 0,Y 502.121,Z 736.307,A -85,B 0,C 180,E1 -5757.593,E2 -5757.593} C_VEL
LIN {X 0,Y 501.992,Z 737.956,A -85,B 0,C 180,E1 -5759.198,E2 -5759.198} C_VEL
LIN {X 0,Y 501.981,Z 738.207,A -85,B 0,C 180,E1 -5760,E2 -5760} C_VEL
LIN {X 0,Y 501.992,Z 738.025,A -85,B 0,C 180,E1 -5760.802,E2 -5760.802} C_VEL
LIN {X 0,Y 502.121,Z 736.475,A -85,B 0,C 180,E1 -5762.406,E2 -5762.406} C_VEL
LIN {X 0,Y 502.125,Z 735.105,A -85,B 0,C 180,E1 -5763.209,E2 -5763.209} C_VEL
LIN {X 0,Y 502.209,Z 732.221,A -85,B 0,C 180,E1 -5764.414,E2 -5764.414} C_VEL
LIN {X 0,Y 502.288,Z 728.294,A -85,B 0,C 180,E1 -5765.621,E2 -5765.621} C_VEL
LIN {X 0,Y 502.401,Z 722.312,A -85,B 0,C 180,E1 -5767.01,E2 -5767.01} C_VEL
LIN {X 0,Y 502.624,Z 715.563,A -85,B 0,C 180,E1 -5768.24,E2 -5768.24} C_VEL
LIN {X 0,Y 502.822,Z 707.24,A -85,B 0,C 180,E1 -5769.452,E2 -5769.452} C_VEL
LIN {X 0,Y 503.101,Z 698.672,A -85,B 0,C 180,E1 -5770.463,E2 -5770.463} C_VEL
LIN {X 0,Y 503.513,Z 688.135,A -85,B 0,C 180,E1 -5771.473,E2 -5771.473} C_VEL
LIN {X 0,Y 503.799,Z 676.957,A -85,B 0,C 180,E1 -5772.322,E2 -5772.322} C_VEL
LIN {X 0,Y 504.044,Z 665.8,A -85,B 0,C 180,E1 -5772.993,E2 -5772.993} C_VEL
LIN {X 0,Y 504.392,Z 653.689,A -85,B 0,C 180,E1 -5773.548,E2 -5773.548} C_VEL
LIN {X 0,Y 504.614,Z 640.164,A -85,B 0,C 180,E1 -5773.978,E2 -5773.978} C_VEL
LIN {X 0,Y 504.768,Z 627.073,A -85,B 0,C 180,E1 -5774.231,E2 -5774.231} C_VEL
LIN {X 0,Y 505.265,Z 535.851,A -85,B 0,C 180,E1 -5775.613,E2 -5775.613} C_VEL
LIN {X 0,Y 503.759,Z 526.619,A -85,B 0,C 180,E1 -5775.813,E2 -5775.813} C_VEL
LIN {X 0,Y 504.19,Z 505.472,A -85,B 0,C 180,E1 -5778.91,E2 -5778.91} C_VEL
LIN {X 0,Y 504.597,Z 484.859,A -85,B 0,C 180,E1 -5781.874,E2 -5781.874} C_VEL
LIN {X 0,Y 504.754,Z 469.617,A -85,B 0,C 180,E1 -5784.033,E2 -5784.033} C_VEL
LIN {X 0,Y 502.898,Z 459.47,A -85,B 0,C 180,E1 -5785.566,E2 -5785.566} C_VEL
LIN {X 0,Y 502.845,Z 459.478,A -85,B 0,C 180,E1 -5788.372,E2 -5788.372} C_VEL
LIN {X 0,Y 502.799,Z 459.48,A -85,B 0,C 180,E1 -5791.499,E2 -5791.499} C_VEL
LIN {X 0,Y 502.811,Z 459.479,A -85,B 0,C 180,E1 -5794.444,E2 -5794.444} C_VEL
LIN {X 0,Y 502.786,Z 459.478,A -85,B 0,C 180,E1 -5797.178,E2 -5797.178} C_VEL
LIN {X 0,Y 502.792,Z 459.482,A -85,B 0,C 180,E1 -5800.015,E2 -5800.015} C_VEL
LIN {X 0,Y 502.807,Z 459.48,A -85,B 0,C 180,E1 -5802.199,E2 -5802.199} C_VEL
LIN {X 0,Y 502.79,Z 459.481,A -85,B 0,C 180,E1 -5805.47,E2 -5805.47} C_VEL
LIN {X 0,Y 502.824,Z 459.473,A -85,B 0,C 180,E1 -5808.934,E2 -5808.934} C_VEL
LIN {X 0,Y 502.797,Z 459.479,A -85,B 0,C 180,E1 -5812.046,E2 -5812.046} C_VEL
LIN {X 0,Y 502.803,Z 459.478,A -85,B 0,C 180,E1 -5815.034,E2 -5815.034} C_VEL
LIN {X 0,Y 502.788,Z 459.482,A -85,B 0,C 180,E1 -5817.915,E2 -5817.915} C_VEL
LIN {X 0,Y 502.829,Z 459.476,A -85,B 0,C 180,E1 -5820.712,E2 -5820.712} C_VEL
LIN {X 0,Y 502.885,Z 459.669,A -85,B 0,C 180,E1 -5822.747,E2 -5822.747} C_VEL
LIN {X 0,Y 506.221,Z 473.456,A -85,B 0,C 180,E1 -5824.735,E2 -5824.735} C_VEL
LIN {X 0,Y 506.3,Z 478.493,A -85,B 0,C 180,E1 -5825.39,E2 -5825.39} C_VEL
LIN {X 0,Y 505.31,Z 502.568,A -85,B 0,C 180,E1 -5828.415,E2 -5828.415} C_VEL
LIN {X 0,Y 504.565,Z 523.078,A -85,B 0,C 180,E1 -5830.963,E2 -5830.963} C_VEL
LIN {X 0,Y 506.669,Z 537.141,A -85,B 0,C 180,E1 -5831.26,E2 -5831.26} C_VEL
LIN {X 0,Y 505.683,Z 661.404,A -85,B 0,C 180,E1 -5833.108,E2 -5833.108} C_VEL
LIN {X 0,Y 505.374,Z 675.938,A -85,B 0,C 180,E1 -5833.488,E2 -5833.488} C_VEL
LIN {X 0,Y 505.054,Z 690.5,A -85,B 0,C 180,E1 -5834.047,E2 -5834.047} C_VEL
LIN {X 0,Y 504.678,Z 702.531,A -85,B 0,C 180,E1 -5834.657,E2 -5834.657} C_VEL
LIN {X 0,Y 504.181,Z 715.296,A -85,B 0,C 180,E1 -5835.468,E2 -5835.468} C_VEL
LIN {X 0,Y 503.724,Z 728.139,A -85,B 0,C 180,E1 -5836.484,E2 -5836.484} C_VEL
LIN {X 0,Y 503.318,Z 738.985,A -85,B 0,C 180,E1 -5837.54,E2 -5837.54} C_VEL
LIN {X 0,Y 502.983,Z 748.981,A -85,B 0,C 180,E1 -5838.718,E2 -5838.718} C_VEL
LIN {X 0,Y 502.66,Z 757.567,A -85,B 0,C 180,E1 -5839.934,E2 -5839.934} C_VEL
LIN {X 0,Y 502.458,Z 764.722,A -85,B 0,C 180,E1 -5841.148,E2 -5841.148} C_VEL
LIN {X 0,Y 502.298,Z 770.625,A -85,B 0,C 180,E1 -5842.361,E2 -5842.361} C_VEL
LIN {X 0,Y 502.215,Z 775.475,A -85,B 0,C 180,E1 -5843.571,E2 -5843.571} C_VEL
LIN {X 0,Y 502.172,Z 779.403,A -85,B 0,C 180,E1 -5844.78,E2 -5844.78} C_VEL
LIN {X 0,Y 502.133,Z 782.414,A -85,B 0,C 180,E1 -5845.986,E2 -5845.986} C_VEL
LIN {X 0,Y 502.118,Z 785.178,A -85,B 0,C 180,E1 -5847.592,E2 -5847.592} C_VEL
LIN {X 0,Y 501.988,Z 786.542,A -85,B 0,C 180,E1 -5849.197,E2 -5849.197} C_VEL
LIN {X 0,Y 501.986,Z 786.543,A -85,B 0,C 180,E1 -5850.801,E2 -5850.801} C_VEL
LIN {X 0,Y 502.117,Z 785.184,A -85,B 0,C 180,E1 -5852.405,E2 -5852.405} C_VEL
LIN {X 0,Y 502.132,Z 782.426,A -85,B 0,C 180,E1 -5854.012,E2 -5854.012} C_VEL
LIN {X 0,Y 502.211,Z 778.197,A -85,B 0,C 180,E1 -5855.621,E2 -5855.621} C_VEL
LIN {X 0,Y 502.252,Z 772.358,A -85,B 0,C 180,E1 -5857.234,E2 -5857.234} C_VEL
LIN {X 0,Y 502.426,Z 765.773,A -85,B 0,C 180,E1 -5858.647,E2 -5858.647} C_VEL
LIN {X 0,Y 502.66,Z 757.581,A -85,B 0,C 180,E1 -5860.064,E2 -5860.064} C_VEL
LIN {X 0,Y 502.986,Z 748.999,A -85,B 0,C 180,E1 -5861.28,E2 -5861.28} C_VEL
LIN {X 0,Y 503.315,Z 739.005,A -85,B 0,C 180,E1 -5862.457,E2 -5862.457} C_VEL
LIN {X 0,Y 503.723,Z 728.163,A -85,B 0,C 180,E1 -5863.514,E2 -5863.514} C_VEL
LIN {X 0,Y 504.129,Z 716.781,A -85,B 0,C 180,E1 -5864.429,E2 -5864.429} C_VEL
LIN {X 0,Y 504.607,Z 704.361,A -85,B 0,C 180,E1 -5865.24,E2 -5865.24} C_VEL
LIN {X 0,Y 505.022,Z 691.678,A -85,B 0,C 180,E1 -5865.9,E2 -5865.9} C_VEL
LIN {X 0,Y 505.344,Z 677.74,A -85,B 0,C 180,E1 -5866.452,E2 -5866.452} C_VEL
LIN {X 0,Y 505.625,Z 663.06,A -85,B 0,C 180,E1 -5866.856,E2 -5866.856} C_VEL
LIN {X 0,Y 505.883,Z 640.122,A -85,B 0,C 180,E1 -5867.221,E2 -5867.221} C_VEL
LIN {X 0,Y 506.613,Z 536.628,A -85,B 0,C 180,E1 -5868.75,E2 -5868.75} C_VEL
LIN {X 0,Y 504.555,Z 523.121,A -85,B 0,C 180,E1 -5869.028,E2 -5869.028} C_VEL
LIN {X 0,Y 505.44,Z 498.851,A -85,B 0,C 180,E1 -5872.049,E2 -5872.049} C_VEL
LIN {X 0,Y 506.369,Z 476.925,A -85,B 0,C 180,E1 -5874.809,E2 -5874.809} C_VEL
LIN {X 0,Y 506.19,Z 473.529,A -85,B 0,C 180,E1 -5875.258,E2 -5875.258} C_VEL
LIN {X 0,Y 502.837,Z 459.475,A -85,B 0,C 180,E1 -5877.307,E2 -5877.307} C_VEL
LIN {X 0,Y 502.816,Z 459.476,A -85,B 0,C 180,E1 -5880.209,E2 -5880.209} C_VEL
LIN {X 0,Y 502.827,Z 459.476,A -85,B 0,C 180,E1 -5883.03,E2 -5883.03} C_VEL
LIN {X 0,Y 502.779,Z 459.474,A -85,B 0,C 180,E1 -5885.949,E2 -5885.949} C_VEL
LIN {X 0,Y 502.816,Z 459.479,A -85,B 0,C 180,E1 -5888.973,E2 -5888.973} C_VEL
LIN {X 0,Y 502.82,Z 459.475,A -85,B 0,C 180,E1 -5892.201,E2 -5892.201} C_VEL
LIN {X 0,Y 502.793,Z 459.475,A -85,B 0,C 180,E1 -5895.467,E2 -5895.467} C_VEL
LIN {X 0,Y 502.821,Z 459.471,A -85,B 0,C 180,E1 -5897.863,E2 -5897.863} C_VEL
LIN {X 0,Y 502.814,Z 459.475,A -85,B 0,C 180,E1 -5901.025,E2 -5901.025} C_VEL
LIN {X 0,Y 502.777,Z 459.472,A -85,B 0,C 180,E1 -5904.166,E2 -5904.166} C_VEL
LIN {X 0,Y 502.823,Z 459.474,A -85,B 0,C 180,E1 -5906.992,E2 -5906.992} C_VEL
LIN {X 0,Y 502.82,Z 459.473,A -85,B 0,C 180,E1 -5910.061,E2 -5910.061} C_VEL
LIN {X 0,Y 502.826,Z 459.476,A -85,B 0,C 180,E1 -5912.533,E2 -5912.533} C_VEL
LIN {X 0,Y 502.818,Z 459.471,A -85,B 0,C 180,E1 -5915.298,E2 -5915.298} C_VEL
LIN {X 0,Y 502.774,Z 459.466,A -85,B 0,C 180,E1 -5917.826,E2 -5917.826} C_VEL
LIN {X 0,Y 502.815,Z 459.473,A -85,B 0,C 180,E1 -5920.4,E2 -5920.4} C_VEL
LIN {X 0,Y 502.826,Z 459.474,A -85,B 0,C 180,E1 -5922.931,E2 -5922.931} C_VEL
LIN {X 0,Y 502.834,Z 459.47,A -85,B 0,C 180,E1 -5925.429,E2 -5925.429} C_VEL
LIN {X 0,Y 502.884,Z 459.468,A -85,B 0,C 180,E1 -5928.717,E2 -5928.717} C_VEL
LIN {X 0,Y 502.891,Z 459.464,A -85,B 0,C 180,E1 -5931.967,E2 -5931.967} C_VEL
LIN {X 0,Y 502.938,Z 459.459,A -85,B 0,C 180,E1 -5934.387,E2 -5934.387} C_VEL
LIN {X 0,Y 503.015,Z 459.446,A -85,B 0,C 180,E1 -5937.598,E2 -5937.598} C_VEL
LIN {X 0,Y 503.016,Z 459.448,A -85,B 0,C 180,E1 -5940,E2 -5940} C_VEL
LIN {X 0,Y 503.015,Z 459.454,A -85,B 0,C 180,E1 -5942.402,E2 -5942.402} C_VEL
LIN {X 0,Y 502.929,Z 459.458,A -85,B 0,C 180,E1 -5945.614,E2 -5945.614} C_VEL
LIN {X 0,Y 502.891,Z 459.463,A -85,B 0,C 180,E1 -5948.034,E2 -5948.034} C_VEL
LIN {X 0,Y 502.884,Z 459.464,A -85,B 0,C 180,E1 -5951.283,E2 -5951.283} C_VEL
LIN {X 0,Y 502.841,Z 459.476,A -85,B 0,C 180,E1 -5954.571,E2 -5954.571} C_VEL
LIN {X 0,Y 502.851,Z 459.467,A -85,B 0,C 180,E1 -5957.908,E2 -5957.908} C_VEL
LIN {X 0,Y 502.818,Z 459.48,A -85,B 0,C 180,E1 -5960.537,E2 -5960.537} C_VEL
LIN {X 0,Y 502.787,Z 459.478,A -85,B 0,C 180,E1 -5963.041,E2 -5963.041} C_VEL
LIN {X 0,Y 502.832,Z 459.47,A -85,B 0,C 180,E1 -5965.676,E2 -5965.676} C_VEL
LIN {X 0,Y 502.833,Z 459.477,A -85,B 0,C 180,E1 -5968.373,E2 -5968.373} C_VEL
LIN {X 0,Y 502.788,Z 459.476,A -85,B 0,C 180,E1 -5971.501,E2 -5971.501} C_VEL
LIN {X 0,Y 502.799,Z 459.48,A -85,B 0,C 180,E1 -5974.446,E2 -5974.446} C_VEL
LIN {X 0,Y 502.774,Z 459.477,A -85,B 0,C 180,E1 -5977.18,E2 -5977.18} C_VEL
LIN {X 0,Y 502.819,Z 459.475,A -85,B 0,C 180,E1 -5980.012,E2 -5980.012} C_VEL
LIN {X 0,Y 502.766,Z 459.479,A -85,B 0,C 180,E1 -5983.232,E2 -5983.232} C_VEL
LIN {X 0,Y 502.784,Z 459.477,A -85,B 0,C 180,E1 -5985.662,E2 -5985.662} C_VEL
LIN {X 0,Y 502.824,Z 459.474,A -85,B 0,C 180,E1 -5987.865,E2 -5987.865} C_VEL
LIN {X 0,Y 502.818,Z 459.475,A -85,B 0,C 180,E1 -5991.027,E2 -5991.027} C_VEL
LIN {X 0,Y 502.782,Z 459.48,A -85,B 0,C 180,E1 -5994.168,E2 -5994.168} C_VEL
LIN {X 0,Y 502.806,Z 459.476,A -85,B 0,C 180,E1 -5997.236,E2 -5997.236} C_VEL
LIN {X 0,Y 502.109,Z 459.566,A -85,B 0,C 180,E1 -5997.905,E2 -5997.905} C_VEL
LIN {X 0,Y 499.251,Z 459.921,A -85,B 0,C 180,E1 -5998.991,E2 -5998.991} C_VEL
LIN {X 0,Y 496.86,Z 460.219,A -85,B 0,C 180,E1 -5999.866,E2 -5999.866} C_VEL
LIN {X 0,Y 495.842,Z 460.347,A -85,B 0,C 180,E1 -6000.541,E2 -6000.541} C_VEL
LIN {X 0,Y 495.763,Z 460.355,A -85,B 0,C 180,E1 -6000.77,E2 -6000.77} C_VEL
LIN {X 0,Y 495.802,Z 460.352,A -85,B 0,C 180,E1 -6003.934,E2 -6003.934} C_VEL
LIN {X 0,Y 495.812,Z 460.431,A -85,B 0,C 180,E1 -6004.414,E2 -6004.414} C_VEL
LIN {X 0,Y 498.119,Z 471.667,A -85,B 0,C 180,E1 -6006.505,E2 -6006.505} C_VEL
LIN {X 0,Y 497.844,Z 483.159,A -85,B 0,C 180,E1 -6008.468,E2 -6008.468} C_VEL
LIN {X 0,Y 497.031,Z 503.536,A -85,B 0,C 180,E1 -6011.877,E2 -6011.877} C_VEL
LIN {X 0,Y 496.68,Z 515.766,A -85,B 0,C 180,E1 -6013.862,E2 -6013.862} C_VEL
LIN {X 0,Y 498.955,Z 528.581,A -85,B 0,C 180,E1 -6014.126,E2 -6014.126} C_VEL
LIN {X 0,Y 498.536,Z 625.651,A -85,B 0,C 180,E1 -6015.484,E2 -6015.484} C_VEL
LIN {X 0,Y 498.317,Z 638.167,A -85,B 0,C 180,E1 -6015.817,E2 -6015.817} C_VEL
LIN {X 0,Y 497.977,Z 651.008,A -85,B 0,C 180,E1 -6016.327,E2 -6016.327} C_VEL
LIN {X 0,Y 497.623,Z 662.342,A -85,B 0,C 180,E1 -6016.941,E2 -6016.941} C_VEL
LIN {X 0,Y 497.18,Z 673.943,A -85,B 0,C 180,E1 -6017.76,E2 -6017.76} C_VEL
LIN {X 0,Y 496.713,Z 684.326,A -85,B 0,C 180,E1 -6018.679,E2 -6018.679} C_VEL
LIN {X 0,Y 496.306,Z 694.518,A -85,B 0,C 180,E1 -6019.806,E2 -6019.806} C_VEL
LIN {X 0,Y 495.927,Z 703.361,A -85,B 0,C 180,E1 -6021.033,E2 -6021.033} C_VEL
LIN {X 0,Y 495.576,Z 710.504,A -85,B 0,C 180,E1 -6022.258,E2 -6022.258} C_VEL
LIN {X 0,Y 495.35,Z 716.238,A -85,B 0,C 180,E1 -6023.484,E2 -6023.484} C_VEL
LIN {X 0,Y 495.142,Z 720.778,A -85,B 0,C 180,E1 -6024.707,E2 -6024.707} C_VEL
LIN {X 0,Y 495.172,Z 724.244,A -85,B 0,C 180,E1 -6025.932,E2 -6025.932} C_VEL
LIN {X 0,Y 495.138,Z 726.04,A -85,B 0,C 180,E1 -6026.746,E2 -6026.746} C_VEL
LIN {X 0,Y 494.963,Z 728.363,A -85,B 0,C 180,E1 -6028.374,E2 -6028.374} C_VEL
LIN {X 0,Y 494.904,Z 729.187,A -85,B 0,C 180,E1 -6030.001,E2 -6030.001} C_VEL
LIN {X 0,Y 494.964,Z 728.444,A -85,B 0,C 180,E1 -6031.628,E2 -6031.628} C_VEL
LIN {X 0,Y 495.11,Z 726.196,A -85,B 0,C 180,E1 -6033.256,E2 -6033.256} C_VEL
LIN {X 0,Y 495.158,Z 723.433,A -85,B 0,C 180,E1 -6034.478,E2 -6034.478} C_VEL
LIN {X 0,Y 495.241,Z 719.689,A -85,B 0,C 180,E1 -6035.702,E2 -6035.702} C_VEL
LIN {X 0,Y 495.439,Z 714.048,A -85,B 0,C 180,E1 -6037.111,E2 -6037.111} C_VEL
LIN {X 0,Y 495.73,Z 707.636,A -85,B 0,C 180,E1 -6038.357,E2 -6038.357} C_VEL
LIN {X 0,Y 496.04,Z 699.797,A -85,B 0,C 180,E1 -6039.584,E2 -6039.584} C_VEL
LIN {X 0,Y 496.364,Z 691.81,A -85,B 0,C 180,E1 -6040.608,E2 -6040.608} C_VEL
LIN {X 0,Y 496.838,Z 682.071,A -85,B 0,C 180,E1 -6041.63,E2 -6041.63} C_VEL
LIN {X 0,Y 497.333,Z 671.546,A -85,B 0,C 180,E1 -6042.515,E2 -6042.515} C_VEL
LIN {X 0,Y 497.667,Z 660.338,A -85,B 0,C 180,E1 -6043.267,E2 -6043.267} C_VEL
LIN {X 0,Y 498.096,Z 648.421,A -85,B 0,C 180,E1 -6043.88,E2 -6043.88} C_VEL
LIN {X 0,Y 498.377,Z 636.162,A -85,B 0,C 180,E1 -6044.34,E2 -6044.34} C_VEL
LIN {X 0,Y 498.583,Z 623.407,A -85,B 0,C 180,E1 -6044.647,E2 -6044.647} C_VEL
LIN {X 0,Y 498.945,Z 528.054,A -85,B 0,C 180,E1 -6045.972,E2 -6045.972} C_VEL
LIN {X 0,Y 496.681,Z 515.637,A -85,B 0,C 180,E1 -6046.231,E2 -6046.231} C_VEL
LIN {X 0,Y 497.252,Z 496.394,A -85,B 0,C 180,E1 -6049.4,E2 -6049.4} C_VEL
LIN {X 0,Y 497.964,Z 479.857,A -85,B 0,C 180,E1 -6052.182,E2 -6052.182} C_VEL
LIN {X 0,Y 498.184,Z 472.07,A -85,B 0,C 180,E1 -6053.512,E2 -6053.512} C_VEL
LIN {X 0,Y 495.817,Z 460.353,A -85,B 0,C 180,E1 -6055.729,E2 -6055.729} C_VEL
LIN {X 0,Y 495.778,Z 460.356,A -85,B 0,C 180,E1 -6058.815,E2 -6058.815} C_VEL
LIN {X 0,Y 495.762,Z 460.362,A -85,B 0,C 180,E1 -6061.726,E2 -6061.726} C_VEL
LIN {X 0,Y 495.775,Z 460.35,A -85,B 0,C 180,E1 -6064.694,E2 -6064.694} C_VEL
LIN {X 0,Y 495.736,Z 460.362,A -85,B 0,C 180,E1 -6067.562,E2 -6067.562} C_VEL
LIN {X 0,Y 495.773,Z 460.35,A -85,B 0,C 180,E1 -6070.7,E2 -6070.7} C_VEL
LIN {X 0,Y 495.741,Z 460.359,A -85,B 0,C 180,E1 -6073.696,E2 -6073.696} C_VEL
LIN {X 0,Y 495.734,Z 460.356,A -85,B 0,C 180,E1 -6076.306,E2 -6076.306} C_VEL
LIN {X 0,Y 495.772,Z 460.352,A -85,B 0,C 180,E1 -6079.3,E2 -6079.3} C_VEL
LIN {X 0,Y 495.737,Z 460.352,A -85,B 0,C 180,E1 -6082.439,E2 -6082.439} C_VEL
LIN {X 0,Y 495.791,Z 460.353,A -85,B 0,C 180,E1 -6085.458,E2 -6085.458} C_VEL
LIN {X 0,Y 495.762,Z 460.353,A -85,B 0,C 180,E1 -6088.364,E2 -6088.364} C_VEL
LIN {X 0,Y 495.793,Z 460.354,A -85,B 0,C 180,E1 -6091.507,E2 -6091.507} C_VEL
LIN {X 0,Y 495.853,Z 460.494,A -85,B 0,C 180,E1 -6094.029,E2 -6094.029} C_VEL
LIN {X 0,Y 498.103,Z 471.728,A -85,B 0,C 180,E1 -6095.847,E2 -6095.847} C_VEL
LIN {X 0,Y 497.701,Z 489.062,A -85,B 0,C 180,E1 -6098.46,E2 -6098.46} C_VEL
LIN {X 0,Y 497.14,Z 510.791,A -85,B 0,C 180,E1 -6101.729,E2 -6101.729} C_VEL
LIN {X 0,Y 496.774,Z 526.183,A -85,B 0,C 180,E1 -6104.032,E2 -6104.032} C_VEL
LIN {X 0,Y 498.551,Z 537.487,A -85,B 0,C 180,E1 -6104.281,E2 -6104.281} C_VEL
LIN {X 0,Y 497.783,Z 635.61,A -85,B 0,C 180,E1 -6105.8,E2 -6105.8} C_VEL
LIN {X 0,Y 497.596,Z 648.618,A -85,B 0,C 180,E1 -6106.159,E2 -6106.159} C_VEL
LIN {X 0,Y 497.299,Z 661.039,A -85,B 0,C 180,E1 -6106.671,E2 -6106.671} C_VEL
LIN {X 0,Y 496.976,Z 673.506,A -85,B 0,C 180,E1 -6107.363,E2 -6107.363} C_VEL
LIN {X 0,Y 496.636,Z 684.576,A -85,B 0,C 180,E1 -6108.159,E2 -6108.159} C_VEL
LIN {X 0,Y 496.248,Z 695.89,A -85,B 0,C 180,E1 -6109.184,E2 -6109.184} C_VEL
LIN {X 0,Y 495.915,Z 704.993,A -85,B 0,C 180,E1 -6110.208,E2 -6110.208} C_VEL
LIN {X 0,Y 495.611,Z 713.798,A -85,B 0,C 180,E1 -6111.437,E2 -6111.437} C_VEL
LIN {X 0,Y 495.388,Z 720.885,A -85,B 0,C 180,E1 -6112.664,E2 -6112.664} C_VEL
LIN {X 0,Y 495.286,Z 726.526,A -85,B 0,C 180,E1 -6113.891,E2 -6113.891} C_VEL
LIN {X 0,Y 495.047,Z 730.945,A -85,B 0,C 180,E1 -6115.114,E2 -6115.114} C_VEL
LIN {X 0,Y 495.17,Z 733.258,A -85,B 0,C 180,E1 -6115.93,E2 -6115.93} C_VEL
LIN {X 0,Y 495.051,Z 735.158,A -85,B 0,C 180,E1 -6116.745,E2 -6116.745} C_VEL
LIN {X 0,Y 495.054,Z 736.622,A -85,B 0,C 180,E1 -6117.559,E2 -6117.559} C_VEL
LIN {X 0,Y 494.912,Z 738.284,A -85,B 0,C 180,E1 -6119.186,E2 -6119.186} C_VEL
LIN {X 0,Y 494.899,Z 738.538,A -85,B 0,C 180,E1 -6120,E2 -6120} C_VEL
LIN {X 0,Y 494.912,Z 738.356,A -85,B 0,C 180,E1 -6120.814,E2 -6120.814} C_VEL
LIN {X 0,Y 495.054,Z 736.802,A -85,B 0,C 180,E1 -6122.441,E2 -6122.441} C_VEL
LIN {X 0,Y 495.051,Z 735.425,A -85,B 0,C 180,E1 -6123.255,E2 -6123.255} C_VEL
LIN {X 0,Y 495.137,Z 732.529,A -85,B 0,C 180,E1 -6124.477,E2 -6124.477} C_VEL
LIN {X 0,Y 495.233,Z 728.581,A -85,B 0,C 180,E1 -6125.701,E2 -6125.701} C_VEL
LIN {X 0,Y 495.344,Z 722.569,A -85,B 0,C 180,E1 -6127.111,E2 -6127.111} C_VEL
LIN {X 0,Y 495.586,Z 715.789,A -85,B 0,C 180,E1 -6128.358,E2 -6128.358} C_VEL
LIN {X 0,Y 495.802,Z 707.409,A -85,B 0,C 180,E1 -6129.588,E2 -6129.588} C_VEL
LIN {X 0,Y 496.102,Z 698.79,A -85,B 0,C 180,E1 -6130.612,E2 -6130.612} C_VEL
LIN {X 0,Y 496.544,Z 688.172,A -85,B 0,C 180,E1 -6131.636,E2 -6131.636} C_VEL
LIN {X 0,Y 496.851,Z 676.894,A -85,B 0,C 180,E1 -6132.497,E2 -6132.497} C_VEL
LIN {X 0,Y 497.122,Z 665.627,A -85,B 0,C 180,E1 -6133.177,E2 -6133.177} C_VEL
LIN {X 0,Y 497.452,Z 653.263,A -85,B 0,C 180,E1 -6133.741,E2 -6133.741} C_VEL
LIN {X 0,Y 497.723,Z 639.425,A -85,B 0,C 180,E1 -6134.176,E2 -6134.176} C_VEL
LIN {X 0,Y 497.852,Z 623.79,A -85,B 0,C 180,E1 -6134.459,E2 -6134.459} C_VEL
LIN {X 0,Y 498.475,Z 536.976,A -85,B 0,C 180,E1 -6135.813,E2 -6135.813} C_VEL
LIN {X 0,Y 496.832,Z 527.046,A -85,B 0,C 180,E1 -6136.031,E2 -6136.031} C_VEL
LIN {X 0,Y 497.264,Z 507.003,A -85,B 0,C 180,E1 -6138.97,E2 -6138.97} C_VEL
LIN {X 0,Y 497.642,Z 489.34,A -85,B 0,C 180,E1 -6141.542,E2 -6141.542} C_VEL
LIN {X 0,Y 497.963,Z 472.483,A -85,B 0,C 180,E1 -6143.94,E2 -6143.94} C_VEL
LIN {X 0,Y 496.76,Z 464.593,A -85,B 0,C 180,E1 -6145.115,E2 -6145.115} C_VEL
LIN {X 0,Y 495.856,Z 460.348,A -85,B 0,C 180,E1 -6145.782,E2 -6145.782} C_VEL
LIN {X 0,Y 495.777,Z 460.357,A -85,B 0,C 180,E1 -6148.814,E2 -6148.814} C_VEL
LIN {X 0,Y 495.761,Z 460.359,A -85,B 0,C 180,E1 -6151.725,E2 -6151.725} C_VEL
LIN {X 0,Y 495.781,Z 460.353,A -85,B 0,C 180,E1 -6154.695,E2 -6154.695} C_VEL
LIN {X 0,Y 495.736,Z 460.359,A -85,B 0,C 180,E1 -6157.561,E2 -6157.561} C_VEL
LIN {X 0,Y 495.771,Z 460.353,A -85,B 0,C 180,E1 -6160.699,E2 -6160.699} C_VEL
LIN {X 0,Y 495.732,Z 460.362,A -85,B 0,C 180,E1 -6164.001,E2 -6164.001} C_VEL
LIN {X 0,Y 495.73,Z 460.358,A -85,B 0,C 180,E1 -6167.116,E2 -6167.116} C_VEL
LIN {X 0,Y 495.763,Z 460.356,A -85,B 0,C 180,E1 -6169.952,E2 -6169.952} C_VEL
LIN {X 0,Y 495.732,Z 460.356,A -85,B 0,C 180,E1 -6172.553,E2 -6172.553} C_VEL
LIN {X 0,Y 495.782,Z 460.356,A -85,B 0,C 180,E1 -6175.456,E2 -6175.456} C_VEL
LIN {X 0,Y 495.76,Z 460.355,A -85,B 0,C 180,E1 -6178.363,E2 -6178.363} C_VEL
LIN {X 0,Y 495.792,Z 460.35,A -85,B 0,C 180,E1 -6181.506,E2 -6181.506} C_VEL
LIN {X 0,Y 495.813,Z 460.49,A -85,B 0,C 180,E1 -6182.454,E2 -6182.454} C_VEL
LIN {X 0,Y 499.507,Z 475.811,A -85,B 0,C 180,E1 -6184.702,E2 -6184.702} C_VEL
LIN {X 0,Y 499.077,Z 488.905,A -85,B 0,C 180,E1 -6186.391,E2 -6186.391} C_VEL
LIN {X 0,Y 497.922,Z 515.551,A -85,B 0,C 180,E1 -6189.768,E2 -6189.768} C_VEL
LIN {X 0,Y 497.654,Z 523.132,A -85,B 0,C 180,E1 -6190.727,E2 -6190.727} C_VEL
LIN {X 0,Y 499.854,Z 537.259,A -85,B 0,C 180,E1 -6191.024,E2 -6191.024} C_VEL
LIN {X 0,Y 498.802,Z 660.379,A -85,B 0,C 180,E1 -6192.89,E2 -6192.89} C_VEL
LIN {X 0,Y 498.501,Z 674.893,A -85,B 0,C 180,E1 -6193.268,E2 -6193.268} C_VEL
LIN {X 0,Y 498.185,Z 688.442,A -85,B 0,C 180,E1 -6193.783,E2 -6193.783} C_VEL
LIN {X 0,Y 497.738,Z 701.472,A -85,B 0,C 180,E1 -6194.437,E2 -6194.437} C_VEL
LIN {X 0,Y 497.224,Z 714.362,A -85,B 0,C 180,E1 -6195.26,E2 -6195.26} C_VEL
LIN {X 0,Y 496.751,Z 726.103,A -85,B 0,C 180,E1 -6196.186,E2 -6196.186} C_VEL
LIN {X 0,Y 496.369,Z 735.87,A -85,B 0,C 180,E1 -6197.114,E2 -6197.114} C_VEL
LIN {X 0,Y 496.062,Z 745.469,A -85,B 0,C 180,E1 -6198.196,E2 -6198.196} C_VEL
LIN {X 0,Y 495.726,Z 754.26,A -85,B 0,C 180,E1 -6199.379,E2 -6199.379} C_VEL
LIN {X 0,Y 495.435,Z 763.055,A -85,B 0,C 180,E1 -6200.816,E2 -6200.816} C_VEL
LIN {X 0,Y 495.215,Z 770.128,A -85,B 0,C 180,E1 -6202.251,E2 -6202.251} C_VEL
LIN {X 0,Y 495.104,Z 776.082,A -85,B 0,C 180,E1 -6203.78,E2 -6203.78} C_VEL
LIN {X 0,Y 495.031,Z 780.043,A -85,B 0,C 180,E1 -6205.112,E2 -6205.112} C_VEL
LIN {X 0,Y 495.035,Z 783.548,A -85,B 0,C 180,E1 -6206.744,E2 -6206.744} C_VEL
LIN {X 0,Y 495.051,Z 784.76,A -85,B 0,C 180,E1 -6207.558,E2 -6207.558} C_VEL
LIN {X 0,Y 494.908,Z 786.132,A -85,B 0,C 180,E1 -6209.185,E2 -6209.185} C_VEL
LIN {X 0,Y 494.906,Z 786.134,A -85,B 0,C 180,E1 -6210.813,E2 -6210.813} C_VEL
LIN {X 0,Y 495.05,Z 784.767,A -85,B 0,C 180,E1 -6212.44,E2 -6212.44} C_VEL
LIN {X 0,Y 495.032,Z 781.991,A -85,B 0,C 180,E1 -6214.069,E2 -6214.069} C_VEL
LIN {X 0,Y 495.124,Z 777.738,A -85,B 0,C 180,E1 -6215.701,E2 -6215.701} C_VEL
LIN {X 0,Y 495.173,Z 771.872,A -85,B 0,C 180,E1 -6217.338,E2 -6217.338} C_VEL
LIN {X 0,Y 495.353,Z 765.253,A -85,B 0,C 180,E1 -6218.772,E2 -6218.772} C_VEL
LIN {X 0,Y 495.614,Z 757.013,A -85,B 0,C 180,E1 -6220.209,E2 -6220.209} C_VEL
LIN {X 0,Y 495.96,Z 748.37,A -85,B 0,C 180,E1 -6221.441,E2 -6221.441} C_VEL
LIN {X 0,Y 496.309,Z 737.89,A -85,B 0,C 180,E1 -6222.678,E2 -6222.678} C_VEL
LIN {X 0,Y 496.739,Z 727.333,A -85,B 0,C 180,E1 -6223.707,E2 -6223.707} C_VEL
LIN {X 0,Y 497.158,Z 715.848,A -85,B 0,C 180,E1 -6224.635,E2 -6224.635} C_VEL
LIN {X 0,Y 497.66,Z 703.3,A -85,B 0,C 180,E1 -6225.458,E2 -6225.458} C_VEL
LIN {X 0,Y 498.152,Z 689.812,A -85,B 0,C 180,E1 -6226.154,E2 -6226.154} C_VEL
LIN {X 0,Y 498.445,Z 675.549,A -85,B 0,C 180,E1 -6226.71,E2 -6226.71} C_VEL
LIN {X 0,Y 498.8,Z 661.122,A -85,B 0,C 180,E1 -6227.093,E2 -6227.093} C_VEL
LIN {X 0,Y 499.847,Z 537.409,A -85,B 0,C 180,E1 -6228.975,E2 -6228.975} C_VEL
LIN {X 0,Y 497.658,Z 523.071,A -85,B 0,C 180,E1 -6229.275,E2 -6229.275} C_VEL
LIN {X 0,Y 498.61,Z 498.684,A -85,B 0,C 180,E1 -6232.368,E2 -6232.368} C_VEL
LIN {X 0,Y 499.594,Z 477.101,A -85,B 0,C 180,E1 -6235.124,E2 -6235.124} C_VEL
LIN {X 0,Y 497.696,Z 468.161,A -85,B 0,C 180,E1 -6236.41,E2 -6236.41} C_VEL
LIN {X 0,Y 495.803,Z 460.35,A -85,B 0,C 180,E1 -6237.601,E2 -6237.601} C_VEL
LIN {X 0,Y 495.754,Z 460.357,A -85,B 0,C 180,E1 -6240.686,E2 -6240.686} C_VEL
LIN {X 0,Y 495.757,Z 460.353,A -85,B 0,C 180,E1 -6243.563,E2 -6243.563} C_VEL
LIN {X 0,Y 495.729,Z 460.358,A -85,B 0,C 180,E1 -6246.542,E2 -6246.542} C_VEL
LIN {X 0,Y 495.786,Z 460.35,A -85,B 0,C 180,E1 -6249.633,E2 -6249.633} C_VEL
LIN {X 0,Y 495.757,Z 460.358,A -85,B 0,C 180,E1 -6252.878,E2 -6252.878} C_VEL
LIN {X 0,Y 495.729,Z 460.355,A -85,B 0,C 180,E1 -6255.998,E2 -6255.998} C_VEL
LIN {X 0,Y 495.76,Z 460.358,A -85,B 0,C 180,E1 -6258.704,E2 -6258.704} C_VEL
LIN {X 0,Y 495.756,Z 460.351,A -85,B 0,C 180,E1 -6261.409,E2 -6261.409} C_VEL
LIN {X 0,Y 495.749,Z 460.348,A -85,B 0,C 180,E1 -6264.462,E2 -6264.462} C_VEL
LIN {X 0,Y 495.76,Z 460.351,A -85,B 0,C 180,E1 -6267.405,E2 -6267.405} C_VEL
LIN {X 0,Y 495.772,Z 460.352,A -85,B 0,C 180,E1 -6270.254,E2 -6270.254} C_VEL
LIN {X 0,Y 495.823,Z 460.345,A -85,B 0,C 180,E1 -6273.248,E2 -6273.248} C_VEL
LIN {X 0,Y 495.741,Z 460.352,A -85,B 0,C 180,E1 -6275.724,E2 -6275.724} C_VEL
LIN {X 0,Y 495.733,Z 460.346,A -85,B 0,C 180,E1 -6278.371,E2 -6278.371} C_VEL
LIN {X 0,Y 495.774,Z 460.354,A -85,B 0,C 180,E1 -6280.971,E2 -6280.971} C_VEL
LIN {X 0,Y 495.77,Z 460.348,A -85,B 0,C 180,E1 -6283.53,E2 -6283.53} C_VEL
LIN {X 0,Y 495.786,Z 460.35,A -85,B 0,C 180,E1 -6286.056,E2 -6286.056} C_VEL
LIN {X 0,Y 495.864,Z 460.343,A -85,B 0,C 180,E1 -6288.555,E2 -6288.555} C_VEL
LIN {X 0,Y 495.863,Z 460.339,A -85,B 0,C 180,E1 -6291.852,E2 -6291.852} C_VEL
LIN {X 0,Y 495.894,Z 460.335,A -85,B 0,C 180,E1 -6294.307,E2 -6294.307} C_VEL
LIN {X 0,Y 495.984,Z 460.322,A -85,B 0,C 180,E1 -6297.564,E2 -6297.564} C_VEL
LIN {X 0,Y 495.987,Z 460.323,A -85,B 0,C 180,E1 -6300,E2 -6300} C_VEL
LIN {X 0,Y 495.984,Z 460.33,A -85,B 0,C 180,E1 -6302.436,E2 -6302.436} C_VEL
LIN {X 0,Y 495.886,Z 460.336,A -85,B 0,C 180,E1 -6305.694,E2 -6305.694} C_VEL
LIN {X 0,Y 495.863,Z 460.34,A -85,B 0,C 180,E1 -6308.148,E2 -6308.148} C_VEL
LIN {X 0,Y 495.858,Z 460.339,A -85,B 0,C 180,E1 -6311.445,E2 -6311.445} C_VEL
LIN {X 0,Y 495.783,Z 460.354,A -85,B 0,C 180,E1 -6314.783,E2 -6314.783} C_VEL
LIN {X 0,Y 495.778,Z 460.347,A -85,B 0,C 180,E1 -6317.319,E2 -6317.319} C_VEL
LIN {X 0,Y 495.768,Z 460.352,A -85,B 0,C 180,E1 -6319.891,E2 -6319.891} C_VEL
LIN {X 0,Y 495.748,Z 460.357,A -85,B 0,C 180,E1 -6322.861,E2 -6322.861} C_VEL
LIN {X 0,Y 495.79,Z 460.35,A -85,B 0,C 180,E1 -6326.068,E2 -6326.068} C_VEL
LIN {X 0,Y 495.771,Z 460.353,A -85,B 0,C 180,E1 -6328.815,E2 -6328.815} C_VEL
LIN {X 0,Y 495.75,Z 460.353,A -85,B 0,C 180,E1 -6331.727,E2 -6331.727} C_VEL
LIN {X 0,Y 495.769,Z 460.357,A -85,B 0,C 180,E1 -6334.697,E2 -6334.697} C_VEL
LIN {X 0,Y 495.726,Z 460.354,A -85,B 0,C 180,E1 -6337.562,E2 -6337.562} C_VEL
LIN {X 0,Y 495.786,Z 460.352,A -85,B 0,C 180,E1 -6340.053,E2 -6340.053} C_VEL
LIN {X 0,Y 495.719,Z 460.36,A -85,B 0,C 180,E1 -6342.884,E2 -6342.884} C_VEL
LIN {X 0,Y 495.731,Z 460.358,A -85,B 0,C 180,E1 -6346.001,E2 -6346.001} C_VEL
LIN {X 0,Y 495.763,Z 460.357,A -85,B 0,C 180,E1 -6348.706,E2 -6348.706} C_VEL
LIN {X 0,Y 495.76,Z 460.353,A -85,B 0,C 180,E1 -6351.411,E2 -6351.411} C_VEL
LIN {X 0,Y 495.754,Z 460.36,A -85,B 0,C 180,E1 -6354.465,E2 -6354.465} C_VEL
LIN {X 0,Y 495.767,Z 460.353,A -85,B 0,C 180,E1 -6357.407,E2 -6357.407} C_VEL
LIN {X 0,Y 495.78,Z 460.356,A -85,B 0,C 180,E1 -6360.256,E2 -6360.256} C_VEL
LIN {X 0,Y 495.763,Z 460.355,A -85,B 0,C 180,E1 -6360.77,E2 -6360.77} C_VEL
LIN {X 0,Y 495.106,Z 460.438,A -85,B 0,C 180,E1 -6361.223,E2 -6361.223} C_VEL
LIN {X 0,Y 492.314,Z 460.788,A -85,B 0,C 180,E1 -6361.932,E2 -6361.932} C_VEL
LIN {X 0,Y 489.487,Z 461.141,A -85,B 0,C 180,E1 -6362.649,E2 -6362.649} C_VEL
LIN {X 0,Y 488.792,Z 461.226,A -85,B 0,C 180,E1 -6363.11,E2 -6363.11} C_VEL
LIN {X 0,Y 488.798,Z 461.348,A -85,B 0,C 180,E1 -6364.163,E2 -6364.163} C_VEL
LIN {X 0,Y 491.232,Z 473.113,A -85,B 0,C 180,E1 -6366.386,E2 -6366.386} C_VEL
LIN {X 0,Y 490.923,Z 484.824,A -85,B 0,C 180,E1 -6368.413,E2 -6368.413} C_VEL
LIN {X 0,Y 490.083,Z 504.995,A -85,B 0,C 180,E1 -6371.827,E2 -6371.827} C_VEL
LIN {X 0,Y 489.721,Z 515.653,A -85,B 0,C 180,E1 -6373.596,E2 -6373.596} C_VEL
LIN {X 0,Y 492.211,Z 529.455,A -85,B 0,C 180,E1 -6373.887,E2 -6373.887} C_VEL
LIN {X 0,Y 491.787,Z 625.346,A -85,B 0,C 180,E1 -6375.228,E2 -6375.228} C_VEL
LIN {X 0,Y 491.569,Z 638.16,A -85,B 0,C 180,E1 -6375.565,E2 -6375.565} C_VEL
LIN {X 0,Y 491.201,Z 651.13,A -85,B 0,C 180,E1 -6376.082,E2 -6376.082} C_VEL
LIN {X 0,Y 490.78,Z 663.363,A -85,B 0,C 180,E1 -6376.756,E2 -6376.756} C_VEL
LIN {X 0,Y 490.314,Z 674.823,A -85,B 0,C 180,E1 -6377.585,E2 -6377.585} C_VEL
LIN {X 0,Y 489.798,Z 685.114,A -85,B 0,C 180,E1 -6378.518,E2 -6378.518} C_VEL
LIN {X 0,Y 489.37,Z 695.203,A -85,B 0,C 180,E1 -6379.66,E2 -6379.66} C_VEL
LIN {X 0,Y 488.946,Z 703.986,A -85,B 0,C 180,E1 -6380.904,E2 -6380.904} C_VEL
LIN {X 0,Y 488.579,Z 711.073,A -85,B 0,C 180,E1 -6382.147,E2 -6382.147} C_VEL
LIN {X 0,Y 488.31,Z 716.762,A -85,B 0,C 180,E1 -6383.389,E2 -6383.389} C_VEL
LIN {X 0,Y 488.086,Z 721.263,A -85,B 0,C 180,E1 -6384.631,E2 -6384.631} C_VEL
LIN {X 0,Y 488.111,Z 724.699,A -85,B 0,C 180,E1 -6385.873,E2 -6385.873} C_VEL
LIN {X 0,Y 488.059,Z 726.477,A -85,B 0,C 180,E1 -6386.699,E2 -6386.699} C_VEL
LIN {X 0,Y 487.893,Z 728.779,A -85,B 0,C 180,E1 -6388.35,E2 -6388.35} C_VEL
LIN {X 0,Y 487.825,Z 729.596,A -85,B 0,C 180,E1 -6390.001,E2 -6390.001} C_VEL
LIN {X 0,Y 487.894,Z 728.858,A -85,B 0,C 180,E1 -6391.652,E2 -6391.652} C_VEL
LIN {X 0,Y 487.998,Z 727.927,A -85,B 0,C 180,E1 -6392.477,E2 -6392.477} C_VEL
LIN {X 0,Y 488.034,Z 726.627,A -85,B 0,C 180,E1 -6393.303,E2 -6393.303} C_VEL
LIN {X 0,Y 488.096,Z 723.886,A -85,B 0,C 180,E1 -6394.543,E2 -6394.543} C_VEL
LIN {X 0,Y 488.192,Z 720.17,A -85,B 0,C 180,E1 -6395.785,E2 -6395.785} C_VEL
LIN {X 0,Y 488.422,Z 714.581,A -85,B 0,C 180,E1 -6397.213,E2 -6397.213} C_VEL
LIN {X 0,Y 488.723,Z 708.221,A -85,B 0,C 180,E1 -6398.477,E2 -6398.477} C_VEL
LIN {X 0,Y 489.08,Z 700.436,A -85,B 0,C 180,E1 -6399.722,E2 -6399.722} C_VEL
LIN {X 0,Y 489.538,Z 690.774,A -85,B 0,C 180,E1 -6400.967,E2 -6400.967} C_VEL
LIN {X 0,Y 490.062,Z 680.627,A -85,B 0,C 180,E1 -6402.003,E2 -6402.003} C_VEL
LIN {X 0,Y 490.538,Z 669.311,A -85,B 0,C 180,E1 -6402.929,E2 -6402.929} C_VEL
LIN {X 0,Y 490.993,Z 657.869,A -85,B 0,C 180,E1 -6403.662,E2 -6403.662} C_VEL
LIN {X 0,Y 491.361,Z 646.103,A -85,B 0,C 180,E1 -6404.232,E2 -6404.232} C_VEL
LIN {X 0,Y 491.656,Z 633.285,A -85,B 0,C 180,E1 -6404.673,E2 -6404.673} C_VEL
LIN {X 0,Y 491.86,Z 621.216,A -85,B 0,C 180,E1 -6404.931,E2 -6404.931} C_VEL
LIN {X 0,Y 492.078,Z 528.259,A -85,B 0,C 180,E1 -6406.224,E2 -6406.224} C_VEL
LIN {X 0,Y 489.722,Z 515.639,A -85,B 0,C 180,E1 -6406.497,E2 -6406.497} C_VEL
LIN {X 0,Y 490.316,Z 497.816,A -85,B 0,C 180,E1 -6409.467,E2 -6409.467} C_VEL
LIN {X 0,Y 491.064,Z 481.263,A -85,B 0,C 180,E1 -6412.289,E2 -6412.289} C_VEL
LIN {X 0,Y 491.303,Z 473.612,A -85,B 0,C 180,E1 -6413.613,E2 -6413.613} C_VEL
LIN {X 0,Y 488.767,Z 461.232,A -85,B 0,C 180,E1 -6415.956,E2 -6415.956} C_VEL
LIN {X 0,Y 488.738,Z 461.234,A -85,B 0,C 180,E1 -6418.696,E2 -6418.696} C_VEL
LIN {X 0,Y 488.699,Z 461.24,A -85,B 0,C 180,E1 -6421.18,E2 -6421.18} C_VEL
LIN {X 0,Y 488.736,Z 461.23,A -85,B 0,C 180,E1 -6424.113,E2 -6424.113} C_VEL
LIN {X 0,Y 488.686,Z 461.236,A -85,B 0,C 180,E1 -6427.159,E2 -6427.159} C_VEL
LIN {X 0,Y 488.724,Z 461.229,A -85,B 0,C 180,E1 -6430.345,E2 -6430.345} C_VEL
LIN {X 0,Y 488.722,Z 461.23,A -85,B 0,C 180,E1 -6432.828,E2 -6432.828} C_VEL
LIN {X 0,Y 488.706,Z 461.235,A -85,B 0,C 180,E1 -6435.976,E2 -6435.976} C_VEL
LIN {X 0,Y 488.713,Z 461.228,A -85,B 0,C 180,E1 -6438.585,E2 -6438.585} C_VEL
LIN {X 0,Y 488.71,Z 461.23,A -85,B 0,C 180,E1 -6440.948,E2 -6440.948} C_VEL
LIN {X 0,Y 488.692,Z 461.239,A -85,B 0,C 180,E1 -6443.869,E2 -6443.869} C_VEL
LIN {X 0,Y 488.745,Z 461.226,A -85,B 0,C 180,E1 -6446.877,E2 -6446.877} C_VEL
LIN {X 0,Y 488.73,Z 461.235,A -85,B 0,C 180,E1 -6449.781,E2 -6449.781} C_VEL
LIN {X 0,Y 488.798,Z 461.222,A -85,B 0,C 180,E1 -6453.057,E2 -6453.057} C_VEL
LIN {X 0,Y 488.81,Z 461.355,A -85,B 0,C 180,E1 -6453.818,E2 -6453.818} C_VEL
LIN {X 0,Y 491.171,Z 472.966,A -85,B 0,C 180,E1 -6455.709,E2 -6455.709} C_VEL
LIN {X 0,Y 490.886,Z 487.53,A -85,B 0,C 180,E1 -6457.925,E2 -6457.925} C_VEL
LIN {X 0,Y 490.231,Z 509.529,A -85,B 0,C 180,E1 -6461.26,E2 -6461.26} C_VEL
LIN {X 0,Y 489.813,Z 526.429,A -85,B 0,C 180,E1 -6463.81,E2 -6463.81} C_VEL
LIN {X 0,Y 491.737,Z 539.142,A -85,B 0,C 180,E1 -6464.084,E2 -6464.084} C_VEL
LIN {X 0,Y 490.881,Z 636.146,A -85,B 0,C 180,E1 -6465.622,E2 -6465.622} C_VEL
LIN {X 0,Y 490.704,Z 648.261,A -85,B 0,C 180,E1 -6465.961,E2 -6465.961} C_VEL
LIN {X 0,Y 490.358,Z 660.878,A -85,B 0,C 180,E1 -6466.479,E2 -6466.479} C_VEL
LIN {X 0,Y 490.044,Z 672.884,A -85,B 0,C 180,E1 -6467.146,E2 -6467.146} C_VEL
LIN {X 0,Y 489.755,Z 683.317,A -85,B 0,C 180,E1 -6467.885,E2 -6467.885} C_VEL
LIN {X 0,Y 489.303,Z 693.9,A -85,B 0,C 180,E1 -6468.819,E2 -6468.819} C_VEL
LIN {X 0,Y 489.004,Z 703.424,A -85,B 0,C 180,E1 -6469.86,E2 -6469.86} C_VEL
